		IF	axis_is_standstill(axis)
			AND digital_actuator_is_inactive(csp_transfer_crosspusher_reject.reject_sact)
			AND (
					ABS(axis_calculated_cam_slave_position_deg - slave_scaling) < 2 (* CHECKS IF THE CALCULATED MOVE IS WITHIN 2 mm's OF THE SLAVE SCALING - MEANING AT LOAD *)
					OR csp_transfer_crosspusher.loader_clear (* VERIFIES THE LOADER IS CLEAR MEANING IN A RETRACTED POSITION *)
				)		
		THEN			
			axis_move_absolute(
				position 		:= axis_calculated_cam_slave_position_deg, 
				velocity 		:= phase_velocity_degps,
				direction		:= AXIS_SHORTEST_WAY,
				acceleration 	:= MOTOR_MAX_ACCELLERATION_DEGPS2/4,
				deceleration 	:= MOTOR_MAX_DECELLERATION_DEGPS2/4, 
				jerk 			:= MOTOR_MAX_JERK_DEGPS3, 
				buffer_mode 	:= AXIS_BUFFER_MODE_BUFFERED,
				CONVERSION_this := axis
				);
		END_IF

		IF axis_is_absolute_moving(axis)
		THEN
			phase_status_next	:=	CSP_TRANSFER_PHASE_STATUS_PHASING;
		END_IF

		
	CSP_TRANSFER_PHASE_STATUS_PHASING:

		IF axis_is_standstill(axis)
		THEN
			phase_status_next	:=	CSP_TRANSFER_CROSSPUSHER_STATUS_PHASED;
		END_IF

		
	CSP_TRANSFER_CROSSPUSHER_STATUS_PHASED:

		IF engage_enable
		THEN
			phase_status_next := CSP_TRANSFER_CROSSPUSHER_PHASE_STATUS_DONE;
		END_IF
		
		
	CSP_TRANSFER_CROSSPUSHER_PHASE_STATUS_DONE:	(* Phase done *)
			
		phase_running := FALSE;
		phase_done := TRUE;				
	
		
	CSP_TRANSFER_CROSSPUSHER_PHASE_STATUS_ERROR:	(* Phase error *)
		IF	phase_running
		THEN
			phase_error := TRUE;
			axis_disable(axis);									
		END_IF
		phase_running := FALSE;
		
		IF	phase_conditions 	
		THEN
			phase_status_next := CSP_TRANSFER_CROSSPUSHER_PHASE_STATUS_START;
		END_IF		
END_CASE


IF 	NOT debug_phase_state_machine
	OR debug_phase_machine_one_step	
THEN
	phase_status := phase_status_next;
END_IF

(* Phasing timeout *)
IF (phase_running
	AND NOT debug_phase_state_machine)
	OR phase_error
THEN
	IF	timer_is_expired(phase_time_out_tmr)
	THEN
		process_message_set(1, phase_status, 0, phase_faulted_aem);
	END_IF
ELSE
	timer_restart(30000, phase_time_out_tmr);
END_IF
END_ACTION

END_PROGRAM

// ---- Application/CSP/Case/Closing/csp_case_closing.TcPOU
(*********************************** G.D S.p.A. - Technical Department ***********************************
============= PROGRAM INFO ============
FOLDER:             TBD
MACHINES INVOLVED:  TBD 

============= DESCRIPTION =============
csp machine declaration

============= REVISIONS ===============
Date		Version	 	Author      	Description             
----------	-------		------------  	--------------------------------------------
2019/04/05 	0000.00	 	M.Grasso		Creation of the PRG

**********************************************************************************************************)
(*$R process_ref := prc; $*)
PROGRAM csp_case_closing
VAR
		
	prc:												process;
	prc_path:											STRING;
	RFID_status:										csp_case_closing_rfid_status_enum;
	RFID_status_next:									csp_case_closing_rfid_status_enum;
	
	Closing_RFID_Check_Complete: 						BOOL := FALSE;
	Closing_Upper_RFID_Check_Req: 						BOOL := FALSE;
	
	(* RFID *)
	check_pos_tolerance:								LREAL := 2;
	rfid_value_to_check: 								BYTE;
	os_rfid_value:										BYTE;
	ls_rfid_value:										BYTE;
	
	
	rfid_value_to_write:								BYTE;
	
	(*OS*)
	os_rfid_input_buffer:								iol_slave_bis00lh_pdo_input;
	os_rfid_input_bitheader_1:							iol_slave_bis00lh_bitheader_input;
	os_rfid_input_bitheader_2:							iol_slave_bis00lh_bitheader_input;
			
	os_rfid_output_buffer:								iol_slave_bis00lh_pdo_output;
	os_rfid_output_bitheader_1:							iol_slave_bis00lh_bitheader_output;
	os_rfid_output_bitheader_2:							iol_slave_bis00lh_bitheader_output;
	os_upper_rfid_read_value: 							BYTE;
	os_lower_rfid_read_value: 							BYTE;
	
	(*LS*)
	ls_rfid_input_buffer:								iol_slave_bis00lh_pdo_input;
	ls_rfid_input_bitheader_1:							iol_slave_bis00lh_bitheader_input;
	ls_rfid_input_bitheader_2:							iol_slave_bis00lh_bitheader_input;
			
	ls_rfid_output_buffer:								iol_slave_bis00lh_pdo_output;
	ls_rfid_output_bitheader_1:							iol_slave_bis00lh_bitheader_output;
	ls_rfid_output_bitheader_2:							iol_slave_bis00lh_bitheader_output;
	ls_upper_rfid_read_value: 							BYTE;
	ls_lower_rfid_read_value: 							BYTE;


	rfid_start_toggle:									BOOL := FALSE;
	rfid_shutdown_toggle:								BOOL := FALSE;
	rfid_write_toggle:									BOOL := FALSE;
	rfid_write_done:									BOOL := FALSE;
	rfid_read_toggle:									BOOL := FALSE;
	rfid_read_done:										BOOL := FALSE;
	rfid_read_success: 									BOOL := FALSE;
	Closing_paddle_rfid_error: 							message;

	RFID_read_write_debug: 								BOOL := FALSE;
	RFID_read_write_one_step: 							BOOL := FALSE;
	
	LS_Lower_RFID_Failed: 								message;
	OS_Lower_RFID_Failed: 								message;
	LS_Upper_RFID_Failed: 								message;
	OS_Upper_RFID_Failed: 								message;
	
	RFID_read_bypass: 									BOOL;	//added 05/17/21 PRS	
	
	OS_Closing_Paddles_cleanout_position:				BOOL := FALSE; (*$P $*)
	ClosingRfidCheckVel:								REAL := 10;
	
END_VAR

VAR CONSTANT
	MOTOR_MAX_VELOCITY_DEGPS:							LREAL := 9600;
	MOTOR_MAX_ACCELLERATION_DEGPS2:						LREAL := 4800;
	MOTOR_MAX_DECELLERATION_DEGPS2:						LREAL := 4800;
	MOTOR_MAX_JERK_DEGPS3:								LREAL := 100000000; 
	MOTOR_MAX_FOLLOWING_ERROR_DEG:						LREAL := 2;
END_VAR

_read_var_input();

_object_manager();

IF NOT objects_running()
THEN
	RETURN;	
END_IF

_read_process_image();

_mode_manager();

_set_runtime_properties();

(********************************* BODY *********************************)
IF csp_main_accuChange.RFID_reader_list_accuchange = CLOSING_PADDLES_READER
THEN
	RFID();
END_IF
IF
	( 
	NOT csp_main_accuChange.RFID_read_write_running
	AND (RFID_status = CSP_CASE_CLOSING_RFID_STATUS_COMPLETE 
	OR RFID_status = CSP_CASE_CLOSING_RFID_STATUS_ERROR) 
	)	
THEN
	RFID_status_next := CSP_CASE_CLOSING_RFID_STATUS_START;
END_IF
IF csp_main_accuChange.RFID_check_request AND Closing_RFID_Check_Complete 
THEN
	Closing_RFID_Check_Complete := FALSE;
END_IF
IF csp_main_accuChange.RFID_writing 
	OR csp_main_accuChange.RFID_reading
THEN
	CASE RFID_status OF
		
		CSP_CASE_CLOSING_RFID_STATUS_START:
		
			rfid_read_done := FALSE;
			rfid_write_done := FALSE;
			
			rfid_value_to_write := csp_main_accuchange.RFID_Setup_write_value;
		
			IF 	machine_is_ready(csp.mch)
			THEN
				axis_enable(csp_case_closing_ls_horizontal.axis);
				axis_enable(csp_case_closing_os_horizontal.axis);
				axis_enable(csp_case_closing_ls_lower.axis);
				axis_enable(csp_case_closing_ls_upper.axis);
				axis_enable(csp_case_closing_os_lower.axis);
				axis_enable(csp_case_closing_os_upper.axis);
				RFID_status_next := CSP_CASE_CLOSING_RFID_STATUS_ENABLED;
			END_IF
			
		CSP_CASE_CLOSING_RFID_STATUS_ENABLED:
			
						
			IF 	axis_is_standstill(csp_case_closing_ls_horizontal.axis)
				AND axis_is_standstill(csp_case_closing_os_horizontal.axis)
				AND axis_is_standstill(csp_case_closing_ls_lower.axis)
				AND axis_is_standstill(csp_case_closing_ls_upper.axis)
				AND axis_is_standstill(csp_case_closing_os_lower.axis)
				AND axis_is_standstill(csp_case_closing_os_upper.axis)
			THEN
				axis_move_absolute(
					position 		:= csp_case_closing_ls_horizontal.accu_safe_pos,
					velocity 		:= ClosingRfidCheckVel,
					direction		:= AXIS_SHORTEST_WAY,
					acceleration 	:= MOTOR_MAX_ACCELLERATION_DEGPS2 / 10,
					deceleration 	:= MOTOR_MAX_DECELLERATION_DEGPS2 / 10,
					jerk 			:= MOTOR_MAX_JERK_DEGPS3, 
					buffer_mode 	:= AXIS_BUFFER_MODE_BUFFERED,
					CONVERSION_this := csp_case_closing_ls_horizontal.axis); 
				axis_move_absolute(
					position 		:= csp_case_closing_os_horizontal.accu_safe_pos,
					velocity 		:= ClosingRfidCheckVel,
					direction		:= AXIS_SHORTEST_WAY,
					acceleration 	:= MOTOR_MAX_ACCELLERATION_DEGPS2 / 10,
					deceleration 	:= MOTOR_MAX_DECELLERATION_DEGPS2 / 10,
					jerk 			:= MOTOR_MAX_JERK_DEGPS3, 
					buffer_mode 	:= AXIS_BUFFER_MODE_BUFFERED,
					CONVERSION_this := csp_case_closing_os_horizontal.axis); 			
			END_IF;				
					
			IF 	axis_is_absolute_moving(csp_case_closing_os_horizontal.axis) 
				AND axis_is_absolute_moving(csp_case_closing_ls_horizontal.axis)
			THEN
				RFID_status_next := CSP_CASE_CLOSING_RFID_STATUS_PADDLES_START;
			END_IF				
		
			
		CSP_CASE_CLOSING_RFID_STATUS_PADDLES_START://requests upper paddle to move to rfid check position
			
			IF 	csp_main_accuChange.closing_horizontal_safe // AND csp_main_accuchange.Case_Motors_Safe_accU
				AND axis_is_standstill(csp_case_closing_ls_horizontal.axis)
				AND axis_is_standstill(csp_case_closing_os_horizontal.axis)
			THEN
				Closing_Upper_RFID_Check_Req := TRUE;
				axis_move_absolute(
					position         := csp_case_closing_os_upper.accu_safe_pos, //highest point of paddle
					velocity         := ClosingRfidCheckVel,
					direction        := AXIS_SHORTEST_WAY,
					acceleration     := MOTOR_MAX_ACCELLERATION_DEGPS2 / 10,
					deceleration     := MOTOR_MAX_DECELLERATION_DEGPS2 / 10,
					jerk             := MOTOR_MAX_JERK_DEGPS3,
					buffer_mode     := AXIS_BUFFER_MODE_BUFFERED,
					CONVERSION_this := csp_case_closing_os_upper.axis);  
					
				axis_move_absolute(
					position         := csp_case_closing_ls_upper.accu_safe_pos, //highest point of paddle
					velocity         := ClosingRfidCheckVel*0.76,
					direction        := AXIS_SHORTEST_WAY,
					acceleration     := MOTOR_MAX_ACCELLERATION_DEGPS2 / 10,
					deceleration     := MOTOR_MAX_DECELLERATION_DEGPS2 / 10,
					jerk             := MOTOR_MAX_JERK_DEGPS3,
					buffer_mode     := AXIS_BUFFER_MODE_BUFFERED,
					CONVERSION_this := csp_case_closing_ls_upper.axis);  
				axis_move_absolute(
					position         := csp_case_closing_os_lower.accu_safe_pos, //lowest point of paddle
					velocity         := ClosingRfidCheckVel,
					direction        := AXIS_SHORTEST_WAY,
					acceleration     := MOTOR_MAX_ACCELLERATION_DEGPS2 / 10,
					deceleration     := MOTOR_MAX_DECELLERATION_DEGPS2 / 10,
					jerk             := MOTOR_MAX_JERK_DEGPS3,
					buffer_mode     := AXIS_BUFFER_MODE_BUFFERED,
					CONVERSION_this := csp_case_closing_os_lower.axis);  
					
				axis_move_absolute(
					position         := csp_case_closing_ls_lower.accu_safe_pos, //lowest point of paddle
					velocity         := ClosingRfidCheckVel,
					direction        := AXIS_SHORTEST_WAY,
					acceleration     := MOTOR_MAX_ACCELLERATION_DEGPS2 / 10,
					deceleration     := MOTOR_MAX_DECELLERATION_DEGPS2 / 10,
					jerk             := MOTOR_MAX_JERK_DEGPS3,
					buffer_mode     := AXIS_BUFFER_MODE_BUFFERED,
					CONVERSION_this := csp_case_closing_ls_lower.axis);
				
				IF 	(axis_is_absolute_moving(csp_case_closing_ls_upper.axis) OR csp_case_closing_ls_upper.in_accu_safe_pos)
					AND (axis_is_absolute_moving(csp_case_closing_os_upper.axis) OR csp_case_closing_os_upper.in_accu_safe_pos)
					AND (axis_is_absolute_moving(csp_case_closing_os_lower.axis) OR csp_case_closing_os_lower.in_accu_safe_pos)
					AND (axis_is_absolute_moving(csp_case_closing_ls_lower.axis) OR csp_case_closing_ls_lower.in_accu_safe_pos)
				THEN
					RFID_status_next := CSP_CASE_CLOSING_RFID_STATUS_VERIFY_AXIS_SAFE_POS;
				END_IF
			END_IF
		
			
		CSP_CASE_CLOSING_RFID_STATUS_VERIFY_AXIS_SAFE_POS:	
		
			IF 	csp_case_closing_ls_upper.in_accu_safe_pos
				AND csp_case_closing_os_upper.in_accu_safe_pos
				AND csp_case_closing_os_lower.in_accu_safe_pos
				AND csp_case_closing_ls_lower.in_accu_safe_pos
				AND axis_is_standstill(csp_case_closing_ls_lower.axis)
				AND axis_is_standstill(csp_case_closing_ls_upper.axis)
				AND axis_is_standstill(csp_case_closing_os_lower.axis)
				AND axis_is_standstill(csp_case_closing_os_upper.axis)
			THEN
				RFID_status_next := CSP_CASE_CLOSING_RFID_STATUS_UPPER_START;
			END_IF
				
		CSP_CASE_CLOSING_RFID_STATUS_UPPER_START:	
					
			axis_move_absolute(
					position         := csp_case_closing_os_upper.RFID_check_pos, 
					velocity         := ClosingRfidCheckVel,
					direction        := AXIS_SHORTEST_WAY,
					acceleration     := MOTOR_MAX_ACCELLERATION_DEGPS2 / 10,
					deceleration     := MOTOR_MAX_DECELLERATION_DEGPS2 / 10,
					jerk             := MOTOR_MAX_JERK_DEGPS3,
					buffer_mode     := AXIS_BUFFER_MODE_BUFFERED,
					CONVERSION_this := csp_case_closing_os_upper.axis);  
					
				axis_move_absolute(
					position         := csp_case_closing_ls_upper.RFID_check_pos,
					velocity         := ClosingRfidCheckVel*0.76,
					direction        := AXIS_SHORTEST_WAY,
					acceleration     := MOTOR_MAX_ACCELLERATION_DEGPS2 / 10,
					deceleration     := MOTOR_MAX_DECELLERATION_DEGPS2 / 10,
					jerk             := MOTOR_MAX_JERK_DEGPS3,
					buffer_mode     := AXIS_BUFFER_MODE_BUFFERED,
					CONVERSION_this := csp_case_closing_ls_upper.axis);  
			IF axis_is_absolute_moving(csp_case_closing_ls_upper.axis) 
				AND axis_is_absolute_moving(csp_case_closing_os_upper.axis) 
			THEN
				RFID_status_next := CSP_CASE_CLOSING_RFID_STATUS_UPPER_VERIFY_AXIS_POS;
			END_IF
			
		CSP_CASE_CLOSING_RFID_STATUS_UPPER_VERIFY_AXIS_POS:
			
			IF 	(ABS(csp_case_closing_ls_upper.axis.actual_modulo_position - csp_case_closing_ls_upper.rfid_check_pos)) < check_pos_tolerance
				AND
				(ABS(csp_case_closing_os_upper.axis.actual_modulo_position - csp_case_closing_os_upper.rfid_check_pos)) < check_pos_tolerance
				THEN
					RFID_status_next := CSP_CASE_CLOSING_RFID_STATUS_UPPER_READ_START;
			END_IF
		
			
		CSP_CASE_CLOSING_RFID_STATUS_UPPER_READ_START: 
		
			IF 	(
					(
						ls_rfid_input_bitheader_1.CP 
						AND ls_rfid_input_bitheader_2.CP
						AND os_rfid_input_bitheader_1.CP 
						AND os_rfid_input_bitheader_2.CP
					)
					OR RFID_read_bypass
				)  //added 05/17/21 PRS
				AND axis_is_standstill(csp_case_closing_ls_upper.axis)
				AND axis_is_standstill(csp_case_closing_os_upper.axis)
			THEN
				rfid_start_toggle := TRUE; 
				rfid_read_toggle := csp_main_accuchange.RFID_reading;
				rfid_write_toggle := csp_main_accuchange.RFID_writing;
				RFID_status_next := SEL(rfid_read_toggle,CSP_CASE_CLOSING_RFID_STATUS_UPPER_RETURN_TO_SAFE_POS,CSP_CASE_CLOSING_RFID_STATUS_UPPER_READ_CHECK_RESULT);
			END_IF
				
					
		CSP_CASE_CLOSING_RFID_STATUS_UPPER_READ_CHECK_RESULT: //wait for successful read and store values
		
			IF 	rfid_read_success
			THEN
				ls_upper_rfid_read_value := ls_rfid_value;
				os_upper_rfid_read_value := os_rfid_value;
				IF 	ls_rfid_value = os_rfid_value
					OR RFID_read_bypass 
				THEN
					rfid_value_to_check := os_rfid_value;
					RFID_status_next := CSP_CASE_CLOSING_RFID_STATUS_UPPER_RETURN_TO_SAFE_POS;					
				END_IF
			END_IF
			
			
		CSP_CASE_CLOSING_RFID_STATUS_UPPER_RETURN_TO_SAFE_POS:
			
				axis_move_absolute(
					position         := csp_case_closing_os_upper.accu_safe_pos, //highest point of paddle
					velocity         := ClosingRfidCheckVel,
					direction        := AXIS_SHORTEST_WAY,
					acceleration     := MOTOR_MAX_ACCELLERATION_DEGPS2 / 10,
					deceleration     := MOTOR_MAX_DECELLERATION_DEGPS2 / 10,
					jerk             := MOTOR_MAX_JERK_DEGPS3,
					buffer_mode     := AXIS_BUFFER_MODE_BUFFERED,
					CONVERSION_this := csp_case_closing_os_upper.axis);  
					
				axis_move_absolute(
					position         := csp_case_closing_ls_upper.accu_safe_pos, //highest point of paddle
					velocity         := ClosingRfidCheckVel*0.76,
					direction        := AXIS_SHORTEST_WAY,
					acceleration     := MOTOR_MAX_ACCELLERATION_DEGPS2 / 10,
					deceleration     := MOTOR_MAX_DECELLERATION_DEGPS2 / 10,
					jerk             := MOTOR_MAX_JERK_DEGPS3,
					buffer_mode     := AXIS_BUFFER_MODE_BUFFERED,
					CONVERSION_this := csp_case_closing_ls_upper.axis); 
					
				IF 	axis_is_absolute_moving(csp_case_closing_ls_upper.axis) 
					AND axis_is_absolute_moving(csp_case_closing_os_upper.axis) 
				THEN
					RFID_status_next := CSP_CASE_CLOSING_RFID_STATUS_UPPER_READ_DONE;
				END_IF						
			
			
		CSP_CASE_CLOSING_RFID_STATUS_UPPER_READ_DONE://upper has been checked, and is clear to return to safe pos. waits until uppers moved back to safe position
		
			IF csp_case_closing_ls_upper.in_accu_safe_pos 
				AND csp_case_closing_os_upper.in_accu_safe_pos
			THEN
				RFID_status_next := CSP_CASE_CLOSING_RFID_STATUS_LOWER_START;
			END_IF
			
		CSP_CASE_CLOSING_RFID_STATUS_LOWER_START:	
					
			axis_move_absolute(
					position         := csp_case_closing_os_LOWER.RFID_check_pos, 
					velocity         := ClosingRfidCheckVel,
					direction        := AXIS_SHORTEST_WAY,
					acceleration     := MOTOR_MAX_ACCELLERATION_DEGPS2 / 10,
					deceleration     := MOTOR_MAX_DECELLERATION_DEGPS2 / 10,
					jerk             := MOTOR_MAX_JERK_DEGPS3,
					buffer_mode     := AXIS_BUFFER_MODE_BUFFERED,
					CONVERSION_this := csp_case_closing_os_lower.axis);  
					
				axis_move_absolute(
					position         := csp_case_closing_ls_lower.RFID_check_pos,
					velocity         := ClosingRfidCheckVel,
					direction        := AXIS_SHORTEST_WAY,
					acceleration     := MOTOR_MAX_ACCELLERATION_DEGPS2 / 10,
					deceleration     := MOTOR_MAX_DECELLERATION_DEGPS2 / 10,
					jerk             := MOTOR_MAX_JERK_DEGPS3,
					buffer_mode      := AXIS_BUFFER_MODE_BUFFERED,
					CONVERSION_this := csp_case_closing_ls_lower.axis);  
				IF axis_is_absolute_moving(csp_case_closing_ls_lower.axis) 
					AND axis_is_absolute_moving(csp_case_closing_os_LOWER.axis) 
				THEN
					RFID_status_next := CSP_CASE_CLOSING_RFID_STATUS_LOWER_VERIFY_AXIS_POS;
				END_IF
				
		CSP_CASE_CLOSING_RFID_STATUS_LOWER_VERIFY_AXIS_POS:
			
			IF 	ABS(csp_case_closing_os_LOWER.axis.actual_modulo_position - csp_case_closing_os_LOWER.rfid_check_pos) < check_pos_tolerance
				AND
				ABS(csp_case_closing_ls_lower.axis.actual_modulo_position - csp_case_closing_ls_lower.rfid_check_pos) < check_pos_tolerance
				
			THEN
				RFID_status_next := CSP_CASE_CLOSING_RFID_STATUS_LOWER_READ_START;
			END_IF
		
			
		CSP_CASE_CLOSING_RFID_STATUS_LOWER_READ_START: 
		
			IF (
					(
						ls_rfid_input_bitheader_1.CP 
						AND ls_rfid_input_bitheader_2.CP
						AND os_rfid_input_bitheader_1.CP 
						AND os_rfid_input_bitheader_2.CP
					)
					OR RFID_read_bypass
				)
				AND axis_is_standstill(csp_case_closing_os_LOWER.axis)
				AND axis_is_standstill(csp_case_closing_ls_LOWER.axis)
			THEN
				rfid_start_toggle := TRUE; 
				rfid_read_toggle := csp_main_accuchange.RFID_reading;
				rfid_write_toggle := csp_main_accuchange.RFID_writing;
				RFID_status_next := SEL(rfid_read_toggle,CSP_CASE_CLOSING_RFID_STATUS_LOWER_RETURN_TO_SAFE_POS,CSP_CASE_CLOSING_RFID_STATUS_LOWER_READ_CHECK_RESULT);
			END_IF
				
					
		CSP_CASE_CLOSING_RFID_STATUS_LOWER_READ_CHECK_RESULT: //wait for successful read and store values
		
			IF rfid_read_success
			THEN
				ls_lower_rfid_read_value := ls_rfid_value;
				os_lower_rfid_read_value := os_rfid_value;
				IF ls_rfid_value = os_rfid_value
				THEN
					rfid_value_to_check := os_rfid_value;
					RFID_status_next := CSP_CASE_CLOSING_RFID_STATUS_LOWER_RETURN_TO_SAFE_POS;
				END_IF
			END_IF
			
		CSP_CASE_CLOSING_RFID_STATUS_LOWER_RETURN_TO_SAFE_POS:
			
				axis_move_absolute(
					position         := csp_case_closing_os_lower.accu_safe_pos, //highest point of paddle
					velocity         := ClosingRfidCheckVel,
					direction        := AXIS_SHORTEST_WAY,
					acceleration     := MOTOR_MAX_ACCELLERATION_DEGPS2 / 10,
					deceleration     := MOTOR_MAX_DECELLERATION_DEGPS2 / 10,
					jerk             := MOTOR_MAX_JERK_DEGPS3,
					buffer_mode     := AXIS_BUFFER_MODE_BUFFERED,
					CONVERSION_this := csp_case_closing_os_lower.axis);  
					
				axis_move_absolute(
					position         := csp_case_closing_ls_lower.accu_safe_pos, //highest point of paddle
					velocity         := ClosingRfidCheckVel,
					direction        := AXIS_SHORTEST_WAY,
					acceleration     := MOTOR_MAX_ACCELLERATION_DEGPS2 / 10,
					deceleration     := MOTOR_MAX_DECELLERATION_DEGPS2 / 10,
					jerk             := MOTOR_MAX_JERK_DEGPS3,
					buffer_mode     := AXIS_BUFFER_MODE_BUFFERED,
					CONVERSION_this := csp_case_closing_ls_lower.axis); 
					
				IF 	axis_is_absolute_moving(csp_case_closing_os_lower.axis) 
					AND axis_is_absolute_moving(csp_case_closing_ls_lower.axis) 
				THEN
					RFID_status_next := CSP_CASE_CLOSING_RFID_STATUS_LOWER_READ_DONE;
				END_IF						
			
			
		CSP_CASE_CLOSING_RFID_STATUS_LOWER_READ_DONE://upper has been checked, and is clear to return to safe pos. waits until uppers moved back to safe position
		
			IF	csp_case_closing_ls_lower.in_accu_safe_pos 
				AND csp_case_closing_os_lower.in_accu_safe_pos
			THEN
				RFID_status_next := SEL(rfid_read_toggle, CSP_CASE_CLOSING_RFID_STATUS_COMPLETE, CSP_CASE_CLOSING_RFID_STATUS_VERIFY_VALUES);
			END_IF
			
		CSP_CASE_CLOSING_RFID_STATUS_VERIFY_VALUES://checks all four paddles rfid value to be equal
		
			IF ls_lower_rfid_read_value = rfid_value_to_check
				AND os_lower_rfid_read_value = rfid_value_to_check
				AND ls_upper_rfid_read_value = rfid_value_to_check
				AND os_upper_rfid_read_value = rfid_value_to_check
			THEN
				RFID_status_next := CSP_CASE_CLOSING_RFID_STATUS_COMPLETE;
			ELSE
				RFID_status_next := CSP_CASE_CLOSING_RFID_STATUS_ERROR;
			END_IF
			
		CSP_CASE_CLOSING_RFID_STATUS_COMPLETE://checks are complete
		
			rfid_write_done := TRUE;
			rfid_read_done := TRUE;			
			Closing_RFID_Check_Complete := TRUE;
			
		
		CSP_CASE_CLOSING_RFID_STATUS_ERROR: //rfid error
		
			rfid_write_done := TRUE;
			rfid_read_done := TRUE;		
			Closing_RFID_Check_Complete :=FALSE;
			//process_message_set(0,0,0,Closing_paddle_rfid_error); (* Moved to csp_main_accuChange *)
			IF ls_lower_rfid_read_value <> rfid_value_to_check
			THEN
				process_message_set(0,0,0,LS_Lower_RFID_Failed);
			ELSIF os_lower_rfid_read_value <> rfid_value_to_check THEN
				process_message_set(0,0,0,OS_Lower_RFID_Failed);
			ELSIF ls_upper_rfid_read_value <> rfid_value_to_check THEN
				process_message_set(0,0,0,LS_Upper_RFID_Failed);
			ELSIF os_upper_rfid_read_value <> rfid_value_to_check THEN
				process_message_set(0,0,0,OS_Upper_RFID_Failed);
			END_IF
			
	END_CASE
END_IF
(* Resets RFID Failed Messages on Reset  *)
IF machine_get_reset_edge(csp.mch)
THEN
	process_message_reset(LS_Lower_RFID_Failed);
	process_message_reset(OS_Lower_RFID_Failed);
	process_message_reset(LS_Upper_RFID_Failed);
	process_message_reset(OS_Upper_RFID_Failed);
END_IF




(* ADVANCES TO NEXT STEP *)
IF 	NOT RFID_read_write_debug
	OR
	RFID_read_write_one_step	
THEN
	RFID_status := RFID_status_next;
	RFID_read_write_one_step := FALSE;
END_IF
(************************************************************************)

_handle_messages();

_write_output();

ACTION _handle_messages:
;
END_ACTION

ACTION _handle_process_test:
;
END_ACTION

ACTION _mode_manager:
IF process_mode_req_is_pending(prc)
THEN
    process_apply_mode_req_first_step(prc);
    CASE process_get_mode(prc) OF
        MODE_TO_ABSENT:
			;
        MODE_TO_INACTIVE:
			;
        MODE_TO_TEST:
			;
        MODE_TO_OPERATIONAL:
			;
    END_CASE
    process_apply_mode_req_second_step(prc);
END_IF
END_ACTION

ACTION _object_manager:
IF objects_initialization()
THEN
	sub_process_init(
		object_name					:= 'csp_case_closing.prc', 
		process						:= csp_case.prc, 
		CONVERSION_this				:= prc);
		
	prc_path 						:= process_get_path(prc);
	
	process_message_init(
        object_name:= CONCAT(prc_path, 'Closing_paddle_rfid_error'),
        behaviour:= MESSAGE_BEHAVIOUR_STATE,
        reset_timeout:= 0,
        disableable:= TRUE,
        individual_reset:= FALSE,
        machine_reaction:= MACHINE_REACTION_NO_STOP, 
        typology:=  MESSAGE_TYPOLOGY_OBLIGATION, 
        process:= prc,
        CONVERSION_this:= Closing_paddle_rfid_error);
		
	process_message_init(
        object_name:= CONCAT(prc_path, 'LS_Lower_RFID_Failed'),
        behaviour:= MESSAGE_BEHAVIOUR_STATE,
        reset_timeout:= 0,
        disableable:= TRUE,
        individual_reset:= FALSE,
        machine_reaction:= MACHINE_REACTION_NORMAL_STOP, 
        typology:=  MESSAGE_TYPOLOGY_ABNORMAL, 
        process:= prc,
        CONVERSION_this:= LS_Lower_RFID_Failed);

	process_message_init(
        object_name:= CONCAT(prc_path, 'OS_Lower_RFID_Failed'),
        behaviour:= MESSAGE_BEHAVIOUR_STATE,
        reset_timeout:= 0,
        disableable:= TRUE,
        individual_reset:= FALSE,
        machine_reaction:= MACHINE_REACTION_NORMAL_STOP, 
        typology:=  MESSAGE_TYPOLOGY_ABNORMAL, 
        process:= prc,
        CONVERSION_this:= OS_Lower_RFID_Failed);
		
	process_message_init(
        object_name:= CONCAT(prc_path, 'LS_Upper_RFID_Failed'),
        behaviour:= MESSAGE_BEHAVIOUR_STATE,
        reset_timeout:= 0,
        disableable:= TRUE,
        individual_reset:= FALSE,
        machine_reaction:= MACHINE_REACTION_NORMAL_STOP, 
        typology:=  MESSAGE_TYPOLOGY_ABNORMAL, 
        process:= prc,
        CONVERSION_this:= LS_Upper_RFID_Failed);

	process_message_init(
        object_name:= CONCAT(prc_path, 'OS_Upper_RFID_Failed'),
        behaviour:= MESSAGE_BEHAVIOUR_STATE,
        reset_timeout:= 0,
        disableable:= TRUE,
        individual_reset:= FALSE,
        machine_reaction:= MACHINE_REACTION_NORMAL_STOP, 
        typology:=  MESSAGE_TYPOLOGY_ABNORMAL,
        process:= prc,
        CONVERSION_this:= OS_Upper_RFID_Failed);
	
END_IF

IF objects_running()
THEN
	process_cycle(prc);
END_IF
END_ACTION

ACTION _read_process_image:
;
END_ACTION

ACTION _read_var_input:
;
END_ACTION

ACTION _set_runtime_properties:
;
END_ACTION

ACTION _write_output:
;
END_ACTION

ACTION RFID:
(* LS *)
ls_rfid_input_bitheader_1.CP := ls_rfid_input_buffer.ByteArr[0].0;
ls_rfid_input_bitheader_1.AA := ls_rfid_input_buffer.ByteArr[0].1;
ls_rfid_input_bitheader_1.AE := ls_rfid_input_buffer.ByteArr[0].2;
ls_rfid_input_bitheader_1.AF := ls_rfid_input_buffer.ByteArr[0].3;
ls_rfid_input_bitheader_1.Bit4 := ls_rfid_input_buffer.ByteArr[0].4;
ls_rfid_input_bitheader_1._TO := ls_rfid_input_buffer.ByteArr[0].5;
ls_rfid_input_bitheader_1.HF := ls_rfid_input_buffer.ByteArr[0].6;
ls_rfid_input_bitheader_1.BB := ls_rfid_input_buffer.ByteArr[0].7;

ls_rfid_input_bitheader_2.CP := ls_rfid_input_buffer.ByteArr[0].0;
ls_rfid_input_bitheader_2.AA := ls_rfid_input_buffer.ByteArr[0].1;
ls_rfid_input_bitheader_2.AE := ls_rfid_input_buffer.ByteArr[0].2;
ls_rfid_input_bitheader_2.AF := ls_rfid_input_buffer.ByteArr[0].3;
ls_rfid_input_bitheader_2.Bit4 := ls_rfid_input_buffer.ByteArr[0].4;
ls_rfid_input_bitheader_2._TO := ls_rfid_input_buffer.ByteArr[0].5;
ls_rfid_input_bitheader_2.HF := ls_rfid_input_buffer.ByteArr[0].6;
ls_rfid_input_bitheader_2.BB := ls_rfid_input_buffer.ByteArr[0].7;

ls_rfid_output_buffer.ByteArr[0].0 := ls_rfid_output_bitheader_1.AV ;
ls_rfid_output_buffer.ByteArr[0].1 := ls_rfid_output_bitheader_1.Bit1;
ls_rfid_output_buffer.ByteArr[0].2 := ls_rfid_output_bitheader_1.GR;
ls_rfid_output_buffer.ByteArr[0].3 := ls_rfid_output_bitheader_1.Bit3;
ls_rfid_output_buffer.ByteArr[0].4 := ls_rfid_output_bitheader_1.Bit4;
ls_rfid_output_buffer.ByteArr[0].5 := ls_rfid_output_bitheader_1.KA;
ls_rfid_output_buffer.ByteArr[0].6 := ls_rfid_output_bitheader_1.TI;
ls_rfid_output_buffer.ByteArr[0].7 := ls_rfid_output_bitheader_1.Bit7;

ls_rfid_output_buffer.ByteArr[9].0 := ls_rfid_output_bitheader_2.AV ;
ls_rfid_output_buffer.ByteArr[9].1 := ls_rfid_output_bitheader_2.Bit1;
ls_rfid_output_buffer.ByteArr[9].2 := ls_rfid_output_bitheader_2.GR;
ls_rfid_output_buffer.ByteArr[9].3 := ls_rfid_output_bitheader_2.Bit3;
ls_rfid_output_buffer.ByteArr[9].4 := ls_rfid_output_bitheader_2.Bit4;
ls_rfid_output_buffer.ByteArr[9].5 := ls_rfid_output_bitheader_2.KA;
ls_rfid_output_buffer.ByteArr[9].6 := ls_rfid_output_bitheader_2.TI;
ls_rfid_output_buffer.ByteArr[9].7 := ls_rfid_output_bitheader_2.Bit7;


(* OS *)
os_rfid_input_bitheader_1.CP := os_rfid_input_buffer.ByteArr[0].0;
os_rfid_input_bitheader_1.AA := os_rfid_input_buffer.ByteArr[0].1;
os_rfid_input_bitheader_1.AE := os_rfid_input_buffer.ByteArr[0].2;
os_rfid_input_bitheader_1.AF := os_rfid_input_buffer.ByteArr[0].3;
os_rfid_input_bitheader_1.Bit4 := os_rfid_input_buffer.ByteArr[0].4;
os_rfid_input_bitheader_1._TO := os_rfid_input_buffer.ByteArr[0].5;
os_rfid_input_bitheader_1.HF := os_rfid_input_buffer.ByteArr[0].6;
os_rfid_input_bitheader_1.BB := os_rfid_input_buffer.ByteArr[0].7;

os_rfid_input_bitheader_2.CP := os_rfid_input_buffer.ByteArr[0].0;
os_rfid_input_bitheader_2.AA := os_rfid_input_buffer.ByteArr[0].1;
os_rfid_input_bitheader_2.AE := os_rfid_input_buffer.ByteArr[0].2;
os_rfid_input_bitheader_2.AF := os_rfid_input_buffer.ByteArr[0].3;
os_rfid_input_bitheader_2.Bit4 := os_rfid_input_buffer.ByteArr[0].4;
os_rfid_input_bitheader_2._TO := os_rfid_input_buffer.ByteArr[0].5;
os_rfid_input_bitheader_2.HF := os_rfid_input_buffer.ByteArr[0].6;
os_rfid_input_bitheader_2.BB := os_rfid_input_buffer.ByteArr[0].7;

os_rfid_output_buffer.ByteArr[0].0 := os_rfid_output_bitheader_1.AV ;
os_rfid_output_buffer.ByteArr[0].1 := os_rfid_output_bitheader_1.Bit1;
os_rfid_output_buffer.ByteArr[0].2 := os_rfid_output_bitheader_1.GR;
os_rfid_output_buffer.ByteArr[0].3 := os_rfid_output_bitheader_1.Bit3;
os_rfid_output_buffer.ByteArr[0].4 := os_rfid_output_bitheader_1.Bit4;
os_rfid_output_buffer.ByteArr[0].5 := os_rfid_output_bitheader_1.KA;
os_rfid_output_buffer.ByteArr[0].6 := os_rfid_output_bitheader_1.TI;
os_rfid_output_buffer.ByteArr[0].7 := os_rfid_output_bitheader_1.Bit7;

os_rfid_output_buffer.ByteArr[9].0 := os_rfid_output_bitheader_2.AV ;
os_rfid_output_buffer.ByteArr[9].1 := os_rfid_output_bitheader_2.Bit1;
os_rfid_output_buffer.ByteArr[9].2 := os_rfid_output_bitheader_2.GR;
os_rfid_output_buffer.ByteArr[9].3 := os_rfid_output_bitheader_2.Bit3;
os_rfid_output_buffer.ByteArr[9].4 := os_rfid_output_bitheader_2.Bit4;
os_rfid_output_buffer.ByteArr[9].5 := os_rfid_output_bitheader_2.KA;
os_rfid_output_buffer.ByteArr[9].6 := os_rfid_output_bitheader_2.TI;
os_rfid_output_buffer.ByteArr[9].7 := os_rfid_output_bitheader_2.Bit7;


IF rfid_start_toggle
THEN
	ls_rfid_output_bitheader_1.GR := FALSE;
	ls_rfid_output_bitheader_1.KA := FALSE;
	ls_rfid_output_bitheader_1.AV := FALSE;
	ls_rfid_output_bitheader_2.GR := FALSE;
	ls_rfid_output_bitheader_2.KA := FALSE;
	ls_rfid_output_bitheader_2.AV := FALSE;
	
	os_rfid_output_bitheader_1.GR := FALSE;
	os_rfid_output_bitheader_1.KA := FALSE;
	os_rfid_output_bitheader_1.AV := FALSE;
	os_rfid_output_bitheader_2.GR := FALSE;
	os_rfid_output_bitheader_2.KA := FALSE;
	os_rfid_output_bitheader_2.AV := FALSE;
	
	rfid_start_toggle := FALSE;
END_IF

IF rfid_shutdown_toggle
THEN
	ls_rfid_output_bitheader_1.KA := TRUE;
	ls_rfid_output_bitheader_2.KA := TRUE;
	
	os_rfid_output_bitheader_1.KA := TRUE;
	os_rfid_output_bitheader_2.KA := TRUE;
		
	IF 	ls_rfid_input_bitheader_1.HF
		AND ls_rfid_input_bitheader_2.HF
	
		AND os_rfid_input_bitheader_1.HF
		AND os_rfid_input_bitheader_2.HF
	
		AND NOT ls_rfid_input_bitheader_1.CP
		AND NOT ls_rfid_input_bitheader_2.CP
	
		AND NOT os_rfid_input_bitheader_1.CP
		AND NOT os_rfid_input_bitheader_2.CP
	THEN
		ls_rfid_output_bitheader_1.KA := FALSE;
		ls_rfid_output_bitheader_2.KA := FALSE;
		
		os_rfid_output_bitheader_1.KA := FALSE;
		os_rfid_output_bitheader_2.KA := FALSE;
		
		rfid_shutdown_toggle := FALSE;
	END_IF	
END_IF

IF rfid_write_toggle //OR i_rfid_write_from_hmi
THEN	
	ls_rfid_output_buffer.ByteArr[1] := 16#0032;
	ls_rfid_output_buffer.ByteArr[2] := 16#00;
	ls_rfid_output_buffer.ByteArr[3] := 16#00;
	ls_rfid_output_buffer.ByteArr[4] := 16#0001;
	ls_rfid_output_buffer.ByteArr[5] := 16#00;
	ls_rfid_output_buffer.ByteArr[6] := rfid_value_to_write;
	
	os_rfid_output_buffer.ByteArr[1] := 16#0032;
	os_rfid_output_buffer.ByteArr[2] := 16#00;
	os_rfid_output_buffer.ByteArr[3] := 16#00;
	os_rfid_output_buffer.ByteArr[4] := 16#0001;
	os_rfid_output_buffer.ByteArr[5] := 16#00;
	os_rfid_output_buffer.ByteArr[6] := rfid_value_to_write;
	
	ls_rfid_output_bitheader_1.AV := TRUE;
	ls_rfid_output_bitheader_2.AV := TRUE;
	
	os_rfid_output_bitheader_1.AV := TRUE;
	os_rfid_output_bitheader_2.AV := TRUE;
	
	IF ls_rfid_input_bitheader_1.AA 
		AND ls_rfid_input_bitheader_2.AA 
		AND ls_rfid_input_bitheader_1.AE
		AND ls_rfid_input_bitheader_2.AE
		
		AND os_rfid_input_bitheader_1.AA 
		AND os_rfid_input_bitheader_2.AA 
		AND os_rfid_input_bitheader_1.AE
		AND os_rfid_input_bitheader_2.AE
	THEN
		ls_rfid_output_bitheader_1.AV := FALSE;
		ls_rfid_output_bitheader_2.AV := FALSE;
		
		os_rfid_output_bitheader_1.AV := FALSE;
		os_rfid_output_bitheader_2.AV := FALSE;
		
		rfid_write_toggle := FALSE;
	END_IF		
END_IF

IF rfid_read_toggle 
THEN
	rfid_read_success := FALSE;	
	ls_rfid_output_buffer.ByteArr[1] := 16#0001;
	ls_rfid_output_buffer.ByteArr[2] := 16#00;
	ls_rfid_output_buffer.ByteArr[3] := 16#00;
	ls_rfid_output_buffer.ByteArr[4] := 16#0001;
	ls_rfid_output_buffer.ByteArr[5] := 16#00;
	
	os_rfid_output_buffer.ByteArr[1] := 16#0001;
	os_rfid_output_buffer.ByteArr[2] := 16#00;
	os_rfid_output_buffer.ByteArr[3] := 16#00;
	os_rfid_output_buffer.ByteArr[4] := 16#0001;
	os_rfid_output_buffer.ByteArr[5] := 16#00;
	
	ls_rfid_output_bitheader_1.AV := TRUE;
	ls_rfid_output_bitheader_2.AV := TRUE;
	ls_rfid_value := 0;
	
	os_rfid_output_bitheader_1.AV := TRUE;
	os_rfid_output_bitheader_2.AV := TRUE;
	os_rfid_value := 0;
	
	IF ls_rfid_input_bitheader_1.AA 
		AND ls_rfid_input_bitheader_2.AA 
		AND ls_rfid_input_bitheader_1.AE
		AND ls_rfid_input_bitheader_2.AE
		
		AND os_rfid_input_bitheader_1.AA 
		AND os_rfid_input_bitheader_2.AA 
		AND os_rfid_input_bitheader_1.AE
		AND os_rfid_input_bitheader_2.AE
	THEN
		// SAVE VALUES IN INPUT BUFFER [1...8] - CHECK WITH BRAND FOR WHAT VALUE SHOULD BE PRESENT
		ls_rfid_value := ls_rfid_input_buffer.ByteArr[1];
		ls_rfid_output_bitheader_1.AV := FALSE;
		ls_rfid_output_bitheader_2.AV := FALSE;
		
		os_rfid_value := os_rfid_input_buffer.ByteArr[1];
		os_rfid_output_bitheader_1.AV := FALSE;
		os_rfid_output_bitheader_2.AV := FALSE;
		
		IF ls_rfid_value <> 0 AND os_rfid_value <> 0
		THEN
			rfid_read_success := TRUE;
		END_IF
		rfid_read_toggle := FALSE;
	END_IF		
END_IF
END_ACTION

END_PROGRAM

// ---- Application/CSP/Case/Main/Drives/csp_case_main_drives.TcPOU

(*********************************** G.D S.p.A. - Technical Department ***********************************
============= PROGRAM INFO ============
FOLDER:             TBD
MACHINES INVOLVED:  TBD 

============= DESCRIPTION =============

============= REVISIONS ===============
Date		Version	 	Author      	Description             
----------	-------		------------  	--------------------------------------------
2019/04/24 	0000.00	 	M.Grasso		Creation of the PRG

**********************************************************************************************************)
(*$R 
	process_ref:= prc; 
$*)
PROGRAM csp_case_main_drives
VAR
	prc:						process;
	prc_path:					STRING;	
	
	PS2000_ps:					power_supply;
	
	SD2100_drv:					soe_drive;
	SD2200_drv:					soe_drive;
	SD2300_drv:					soe_drive;
	SD2400_drv:					soe_drive;
	SD2500_drv:					soe_drive;
	
	SD12000_drv:				soe_drive;
	SD8000_drv:					soe_drive;
	SD8100_drv:					soe_drive;
	SD8200_drv:					soe_drive;
	SD8300_drv:					soe_drive;
	SD8400_drv:					soe_drive;
	SD8500_drv:					soe_drive;
	SD8600_drv:					soe_drive;
	
	SD10000_drv:				soe_drive;
	SD10100_drv:				soe_drive;
	SD10200_drv:				soe_drive;
	SD10300_drv:				soe_drive;
	SD10400_drv:				soe_drive;
	SD11000_drv:				soe_drive;
	
	SD15000_drv:				soe_drive;
	
	SD26000_drv:				soe_drive;
	SD26100_drv:				soe_drive;
	
END_VAR

VAR CONSTANT
	INCOHERENCE_TIMEOUT_MS:		DINT := 2000;
END_VAR

_read_var_input();

_objects_manager();

IF NOT objects_running()
THEN
	RETURN;	
END_IF

_read_process_image();

_mode_manager();

CASE process_get_mode(prc) OF
	MODE_ABSENT,
	MODE_INACTIVE:
		RETURN;
	MODE_TEST:
		;
END_CASE

_set_runtime_properties();

(********************************* BODY *********************************)

(************************************************************************)

_handle_messages();

_write_output();

ACTION _handle_messages:
;
END_ACTION

ACTION _handle_process_test:
;
END_ACTION

ACTION _mode_manager:
IF process_mode_req_is_pending(prc)
THEN
    process_apply_mode_req_first_step(prc);
    CASE process_get_mode(prc) OF
        MODE_TO_ABSENT:
			;
        MODE_TO_INACTIVE:
			;
        MODE_TO_TEST:
			;
        MODE_TO_OPERATIONAL:
			;
    END_CASE
    process_apply_mode_req_second_step(prc);
END_IF
END_ACTION

ACTION _objects_manager:
IF objects_initialization()
THEN
	sub_process_init(
		object_name					:= 'csp_case_main_drives.prc', 
		process						:= csp_case_main.prc, 
		CONVERSION_this				:= prc);
		
	prc_path 						:= process_get_path(prc);

	(* PS2000 POWER SUPPLY *)
	power_supply_init(
		object_name					:= CONCAT(prc_path, '_PS2000_ps'), 
		vendor						:= DRIVE_BOSCH_REXROTH, 
		process						:= prc, 
		CONVERSION_this				:= PS2000_ps);
		
	power_supply_add_safety_integrated_series(
		safety_integrated_series	:= csp_case_main_safety_drives_PS2000.sis, 
		CONVERSION_this				:= PS2000_ps);		

		(* SD2100 *)
	soe_drive_double_channel_init(
		object_name					:= CONCAT(prc_path, '_SD2100_drv'), 
		device_name					:= 'SD2100', 
		vendor						:= DRIVE_BOSCH_REXROTH, 
		standalone					:= FALSE, 
		channel_a_name				:= 'csp_case_transport_os_leading_axis', 
		channel_b_name				:= 'csp_case_transport_os_trailing_axis', 
		ethercat_master				:= csp_main.cabinet_ethercat_master, 
		process						:= prc, 
		CONVERSION_this				:= SD2100_drv);	
		
	soe_drive_add_power_supply(
		power_supply				:= PS2000_ps, 
		CONVERSION_this				:= SD2100_drv);
		
	IF 	SD2100_drv.channel_a.has_channel
	THEN	
		soe_drive_enable_fsoe(
			handler						:= BOSCH_DRIVE_CHANNEL_A, 
			incoherence_timeout			:= INCOHERENCE_TIMEOUT_MS, 
			connection_interface		:= csp_case_main_safety_interface._SD2100_drv_ChA, 
			group						:= csp_case_main_safety_drives_SD2100.sig, 
			CONVERSION_this				:= SD2100_drv);
	END_IF
		
	IF 	SD2100_drv.channel_B.has_channel
	THEN	
		soe_drive_enable_fsoe(
			handler						:= BOSCH_DRIVE_CHANNEL_B, 
			incoherence_timeout			:= INCOHERENCE_TIMEOUT_MS, 
			connection_interface		:= csp_case_main_safety_interface._SD2100_drv_ChB, 
			group						:= csp_case_main_safety_drives_SD2100.sig, 
			CONVERSION_this				:= SD2100_drv);
	END_IF
	
	(* SD2200 *)
	soe_drive_double_channel_init(
		object_name					:= CONCAT(prc_path, '_SD2200_drv'), 
		device_name					:= 'SD2200', 
		vendor						:= DRIVE_BOSCH_REXROTH, 
		standalone					:= FALSE, 
		channel_a_name				:= 'csp_case_transport_ls_leading_axis', 
		channel_b_name				:= 'csp_case_transport_ls_trailing_axis', 
		ethercat_master				:= csp_main.cabinet_ethercat_master, 
		process						:= prc, 
		CONVERSION_this				:= SD2200_drv);	
		
	soe_drive_add_power_supply(
		power_supply				:= PS2000_ps, 
		CONVERSION_this				:= SD2200_drv);
		
	IF 	SD2200_drv.channel_a.has_channel
	THEN	
		soe_drive_enable_fsoe(
			handler						:= BOSCH_DRIVE_CHANNEL_A, 
			incoherence_timeout			:= INCOHERENCE_TIMEOUT_MS, 
			connection_interface		:= csp_case_main_safety_interface._SD2200_drv_ChA, 
			group						:= csp_case_main_safety_drives_SD2200.sig, 
			CONVERSION_this				:= SD2200_drv);
	END_IF
		
	IF 	SD2200_drv.channel_B.has_channel
	THEN	
		soe_drive_enable_fsoe(
			handler						:= BOSCH_DRIVE_CHANNEL_B, 
			incoherence_timeout			:= INCOHERENCE_TIMEOUT_MS, 
			connection_interface		:= csp_case_main_safety_interface._SD2200_drv_ChB, 
			group						:= csp_case_main_safety_drives_SD2200.sig, 
			CONVERSION_this				:= SD2200_drv);
	END_IF
	
	(* SD2300 *)
	soe_drive_double_channel_init(
		object_name					:= CONCAT(prc_path, '_SD2300_drv'), 
		device_name					:= 'SD2300', 
		vendor						:= DRIVE_BOSCH_REXROTH, 
		standalone					:= FALSE, 
		channel_a_name				:= 'csp_case_closing_os_upper_axis', 
		channel_b_name				:= 'csp_case_closing_os_lower_axis', 
		ethercat_master				:= csp_main.cabinet_ethercat_master, 
		process						:= prc, 
		CONVERSION_this				:= SD2300_drv);	
		
	soe_drive_add_power_supply(
		power_supply				:= PS2000_ps, 
		CONVERSION_this				:= SD2300_drv);
		
	IF 	SD2300_drv.channel_a.has_channel
	THEN	
		soe_drive_enable_fsoe(
			handler						:= BOSCH_DRIVE_CHANNEL_A, 
			incoherence_timeout			:= INCOHERENCE_TIMEOUT_MS, 
			connection_interface		:= csp_case_main_safety_interface._SD2300_drv_ChA, 
			group						:= csp_case_main_safety_drives_SD2300.sig, 
			CONVERSION_this				:= SD2300_drv);
	END_IF
		
	IF 	SD2300_drv.channel_B.has_channel
	THEN	
		soe_drive_enable_fsoe(
			handler						:= BOSCH_DRIVE_CHANNEL_B, 
			incoherence_timeout			:= INCOHERENCE_TIMEOUT_MS, 
			connection_interface		:= csp_case_main_safety_interface._SD2300_drv_ChB, 
			group						:= csp_case_main_safety_drives_SD2300.sig, 
			CONVERSION_this				:= SD2300_drv);
	END_IF
	
	(* SD2400 *)
	soe_drive_double_channel_init(
		object_name					:= CONCAT(prc_path, '_SD2400_drv'), 
		device_name					:= 'SD2400', 
		vendor						:= DRIVE_BOSCH_REXROTH, 
		standalone					:= FALSE, 
		channel_a_name				:= 'csp_case_closing_os_horizontal_axis', 
		channel_b_name				:= 'csp_case_closing_ls_upper_axis', 
		ethercat_master				:= csp_main.cabinet_ethercat_master, 
		process						:= prc, 
		CONVERSION_this				:= SD2400_drv);	
		
	soe_drive_add_power_supply(
		power_supply				:= PS2000_ps, 
		CONVERSION_this				:= SD2400_drv);
		
	IF 	SD2400_drv.channel_a.has_channel
	THEN	
		soe_drive_enable_fsoe(
			handler						:= BOSCH_DRIVE_CHANNEL_A, 
			incoherence_timeout			:= INCOHERENCE_TIMEOUT_MS, 
			connection_interface		:= csp_case_main_safety_interface._SD2400_drv_ChA, 
			group						:= csp_case_main_safety_drives_SD2400.sig, 
			CONVERSION_this				:= SD2400_drv);
	END_IF
		
	IF 	SD2400_drv.channel_B.has_channel
	THEN	
		soe_drive_enable_fsoe(
			handler						:= BOSCH_DRIVE_CHANNEL_B, 
			incoherence_timeout			:= INCOHERENCE_TIMEOUT_MS, 
			connection_interface		:= csp_case_main_safety_interface._SD2400_drv_ChB, 
			group						:= csp_case_main_safety_drives_SD2400.sig, 
			CONVERSION_this				:= SD2400_drv);
	END_IF
	
	(* SD2500 *)
	soe_drive_double_channel_init(
		object_name					:= CONCAT(prc_path, '_SD2500_drv'), 
		device_name					:= 'SD2500', 
		vendor						:= DRIVE_BOSCH_REXROTH, 
		standalone					:= FALSE, 
		channel_a_name				:= 'csp_case_closing_ls_lower_axis', 
		channel_b_name				:= 'csp_case_closing_ls_horizontal_axis', 
		ethercat_master				:= csp_main.cabinet_ethercat_master, 
		process						:= prc, 
		CONVERSION_this				:= SD2500_drv);	
		
	soe_drive_add_power_supply(
		power_supply				:= PS2000_ps, 
		CONVERSION_this				:= SD2500_drv);
		
	IF 	SD2500_drv.channel_a.has_channel
	THEN	
		soe_drive_enable_fsoe(
			handler						:= BOSCH_DRIVE_CHANNEL_A, 
			incoherence_timeout			:= INCOHERENCE_TIMEOUT_MS, 
			connection_interface		:= csp_case_main_safety_interface._SD2500_drv_ChA, 
			group						:= csp_case_main_safety_drives_SD2500.sig, 
			CONVERSION_this				:= SD2500_drv);
	END_IF
		
	IF 	SD2500_drv.channel_B.has_channel
	THEN	
		soe_drive_enable_fsoe(
			handler						:= BOSCH_DRIVE_CHANNEL_B, 
			incoherence_timeout			:= INCOHERENCE_TIMEOUT_MS, 
			connection_interface		:= csp_case_main_safety_interface._SD2500_drv_ChB, 
			group						:= csp_case_main_safety_drives_SD2500.sig, 
			CONVERSION_this				:= SD2500_drv);
	END_IF
	
		
		(* SD12000 *)
	soe_drive_double_channel_init(
		object_name					:= CONCAT(prc_path, '_SD12000_drv'), 
		device_name					:= 'SD12000', 
		vendor						:= DRIVE_BOSCH_REXROTH, 
		standalone					:= FALSE, 
		channel_a_name				:= 'csp_case_discharge_speedBelt_os_axis', 
		channel_b_name				:= 'csp_case_discharge_speedBelt_ls_axis', 
		ethercat_master				:= csp_main.cabinet_ethercat_master, 
		process						:= prc, 
		CONVERSION_this				:= SD12000_drv);	
		
	soe_drive_add_power_supply(
		power_supply				:= PS2000_ps, 
		CONVERSION_this				:= SD12000_drv);
		
	IF 	SD12000_drv.channel_a.has_channel
	THEN	
		soe_drive_enable_fsoe(
			handler						:= BOSCH_DRIVE_CHANNEL_A, 
			incoherence_timeout			:= INCOHERENCE_TIMEOUT_MS, 
			connection_interface		:= csp_case_main_safety_interface._SD12000_drv_ChA, 
			group						:= csp_case_main_safety_drives_SD12000.sig, 
			CONVERSION_this				:= SD12000_drv);
	END_IF
		
	IF 	SD12000_drv.channel_B.has_channel
	THEN	
		soe_drive_enable_fsoe(
			handler						:= BOSCH_DRIVE_CHANNEL_B, 
			incoherence_timeout			:= INCOHERENCE_TIMEOUT_MS, 
			connection_interface		:= csp_case_main_safety_interface._SD12000_drv_ChB, 
			group						:= csp_case_main_safety_drives_SD12000.sig, 
			CONVERSION_this				:= SD12000_drv);
	END_IF
	
	(* SD8000 *)
	soe_drive_double_channel_init(
		object_name					:= CONCAT(prc_path, '_SD8000_drv'), 
		device_name					:= 'SD8000', 
		vendor						:= DRIVE_BOSCH_REXROTH, 
		standalone					:= FALSE, 
		channel_a_name				:= 'csp_case_feed_shuttle_horizontal_axis', 
		channel_b_name				:= 'csp_case_feed_shuttle_vertical_axis', 
		ethercat_master				:= csp_main.cabinet_ethercat_master, 
		process						:= prc, 
		CONVERSION_this				:= SD8000_drv);	
		
	soe_drive_add_power_supply(
		power_supply				:= PS2000_ps, 
		CONVERSION_this				:= SD8000_drv);
		
	IF 	SD8000_drv.channel_a.has_channel
	THEN	
		soe_drive_enable_fsoe(
			handler						:= BOSCH_DRIVE_CHANNEL_A, 
			incoherence_timeout			:= INCOHERENCE_TIMEOUT_MS, 
			connection_interface		:= csp_case_main_safety_interface._SD8000_drv_ChA, 
			group						:= csp_case_main_safety_drives_SD8000.sig, 
			CONVERSION_this				:= SD8000_drv);
	END_IF
		
	IF 	SD8000_drv.channel_B.has_channel
	THEN	
		soe_drive_enable_fsoe(
			handler						:= BOSCH_DRIVE_CHANNEL_B, 
			incoherence_timeout			:= INCOHERENCE_TIMEOUT_MS, 
			connection_interface		:= csp_case_main_safety_interface._SD8000_drv_ChB, 
			group						:= csp_case_main_safety_drives_SD8000.sig, 
			CONVERSION_this				:= SD8000_drv);
	END_IF
	
	(* SD8100 *)
	soe_drive_double_channel_init(
		object_name					:= CONCAT(prc_path, '_SD8100_drv'), 
		device_name					:= 'SD8100', 
		vendor						:= DRIVE_BOSCH_REXROTH, 
		standalone					:= FALSE, 
		channel_a_name				:= 'csp_case_feed_arm_shoulder_axis', 
		channel_b_name				:= 'csp_case_fc_ls_lower_trailingCloser_axis', 
		ethercat_master				:= csp_main.cabinet_ethercat_master, 
		process						:= prc, 
		CONVERSION_this				:= SD8100_drv);	
		
	soe_drive_add_power_supply(
		power_supply				:= PS2000_ps, 
		CONVERSION_this				:= SD8100_drv);
		
	IF 	SD8100_drv.channel_a.has_channel
	THEN	
		soe_drive_enable_fsoe(
			handler						:= BOSCH_DRIVE_CHANNEL_A, 
			incoherence_timeout			:= INCOHERENCE_TIMEOUT_MS, 
			connection_interface		:= csp_case_main_safety_interface._SD8100_drv_ChA, 
			group						:= csp_case_main_safety_drives_SD8100.sig, 
			CONVERSION_this				:= SD8100_drv);
	END_IF
		
	IF 	SD8100_drv.channel_B.has_channel
	THEN	
		soe_drive_enable_fsoe(
			handler						:= BOSCH_DRIVE_CHANNEL_B, 
			incoherence_timeout			:= INCOHERENCE_TIMEOUT_MS, 
			connection_interface		:= csp_case_main_safety_interface._SD8100_drv_ChB, 
			group						:= csp_case_main_safety_drives_SD8100.sig, 
			CONVERSION_this				:= SD8100_drv);
	END_IF	
	
	(* SD8200 *)
	soe_drive_double_channel_init(
		object_name					:= CONCAT(prc_path, '_SD8200_drv'), 
		device_name					:= 'SD8200', 
		vendor						:= DRIVE_BOSCH_REXROTH, 
		standalone					:= FALSE, 
		channel_a_name				:= 'csp_case_feed_arm_elbow_axis', 
		channel_b_name				:= 'csp_case_loader_guide_upstream_axis', 
		ethercat_master				:= csp_main.cabinet_ethercat_master, 
		process						:= prc, 
		CONVERSION_this				:= SD8200_drv);	
		
	soe_drive_add_power_supply(
		power_supply				:= PS2000_ps, 
		CONVERSION_this				:= SD8200_drv);
		
	IF 	SD8200_drv.channel_a.has_channel
	THEN	
		soe_drive_enable_fsoe(
			handler						:= BOSCH_DRIVE_CHANNEL_A, 
			incoherence_timeout			:= INCOHERENCE_TIMEOUT_MS, 
			connection_interface		:= csp_case_main_safety_interface._SD8200_drv_ChA, 
			group						:= csp_case_main_safety_drives_SD8200.sig, 
			CONVERSION_this				:= SD8200_drv);
	END_IF
		
	IF 	SD8200_drv.channel_B.has_channel
	THEN	
		soe_drive_enable_fsoe(
			handler						:= BOSCH_DRIVE_CHANNEL_B, 
			incoherence_timeout			:= INCOHERENCE_TIMEOUT_MS, 
			connection_interface		:= csp_case_main_safety_interface._SD8200_drv_ChB, 
			group						:= csp_case_main_safety_drives_SD8200.sig, 
			CONVERSION_this				:= SD8200_drv);
	END_IF	
	
	(* SD8300 *)
	soe_drive_double_channel_init(
		object_name					:= CONCAT(prc_path, '_SD8300_drv'), 
		device_name					:= 'SD8300', 
		vendor						:= DRIVE_BOSCH_REXROTH, 
		standalone					:= FALSE, 
		channel_a_name				:= 'csp_case_feed_arm_wrist_axis', 
		channel_b_name				:= 'csp_case_loader_guide_downstream_axis', 
		ethercat_master				:= csp_main.cabinet_ethercat_master, 
		process						:= prc, 
		CONVERSION_this				:= SD8300_drv);	
		
	soe_drive_add_power_supply(
		power_supply				:= PS2000_ps, 
		CONVERSION_this				:= SD8300_drv);
		
	IF 	SD8300_drv.channel_a.has_channel
	THEN	
		soe_drive_enable_fsoe(
			handler						:= BOSCH_DRIVE_CHANNEL_A, 
			incoherence_timeout			:= INCOHERENCE_TIMEOUT_MS, 
			connection_interface		:= csp_case_main_safety_interface._SD8300_drv_ChA, 
			group						:= csp_case_main_safety_drives_SD8300.sig, 
			CONVERSION_this				:= SD8300_drv);
	END_IF
		
	IF 	SD8300_drv.channel_B.has_channel
	THEN	
		soe_drive_enable_fsoe(
			handler						:= BOSCH_DRIVE_CHANNEL_B, 
			incoherence_timeout			:= INCOHERENCE_TIMEOUT_MS, 
			connection_interface		:= csp_case_main_safety_interface._SD8300_drv_ChB, 
			group						:= csp_case_main_safety_drives_SD8300.sig, 
			CONVERSION_this				:= SD8300_drv);
	END_IF	
	
	(* SD8400 *)
	soe_drive_double_channel_init(
		object_name					:= CONCAT(prc_path, '_SD8400_drv'), 
		device_name					:= 'SD8400', 
		vendor						:= DRIVE_BOSCH_REXROTH, 
		standalone					:= FALSE, 
		channel_a_name				:= 'csp_case_feed_magazine_os_belt_axis', 
		channel_b_name				:= 'csp_case_feed_magazine_ls_belt_axis', 
		ethercat_master				:= csp_main.cabinet_ethercat_master, 
		process						:= prc, 
		CONVERSION_this				:= SD8400_drv);	
		
	soe_drive_add_power_supply(
		power_supply				:= PS2000_ps, 
		CONVERSION_this				:= SD8400_drv);
		
	IF 	SD8400_drv.channel_a.has_channel
	THEN	
		soe_drive_enable_fsoe(
			handler						:= BOSCH_DRIVE_CHANNEL_A, 
			incoherence_timeout			:= INCOHERENCE_TIMEOUT_MS, 
			connection_interface		:= csp_case_main_safety_interface._SD8400_drv_ChA, 
			group						:= csp_case_main_safety_drives_SD8400.sig, 
			CONVERSION_this				:= SD8400_drv);
	END_IF
		
	IF 	SD8400_drv.channel_B.has_channel
	THEN	
		soe_drive_enable_fsoe(
			handler						:= BOSCH_DRIVE_CHANNEL_B, 
			incoherence_timeout			:= INCOHERENCE_TIMEOUT_MS, 
			connection_interface		:= csp_case_main_safety_interface._SD8400_drv_ChB, 
			group						:= csp_case_main_safety_drives_SD8400.sig, 
			CONVERSION_this				:= SD8400_drv);
	END_IF	
	
	(* SD8500 *)
	soe_drive_double_channel_init(
		object_name					:= CONCAT(prc_path, '_SD8500_drv'), 
		device_name					:= 'SD8500', 
		vendor						:= DRIVE_BOSCH_REXROTH, 
		standalone					:= FALSE, 
		channel_a_name				:= 'csp_case_loader_pusher_axis', 
		channel_b_name				:= 'csp_case_loader_guide_length_axis', 
		ethercat_master				:= csp_main.cabinet_ethercat_master, 
		process						:= prc, 
		CONVERSION_this				:= SD8500_drv);	
		
	soe_drive_add_power_supply(
		power_supply				:= PS2000_ps, 
		CONVERSION_this				:= SD8500_drv);
		
	IF 	SD8500_drv.channel_a.has_channel
	THEN	
		soe_drive_enable_fsoe(
			handler						:= BOSCH_DRIVE_CHANNEL_A, 
			incoherence_timeout			:= INCOHERENCE_TIMEOUT_MS, 
			connection_interface		:= csp_case_main_safety_interface._SD8500_drv_ChA, 
			group						:= csp_case_main_safety_drives_SD8500.sig, 
			CONVERSION_this				:= SD8500_drv);
	END_IF
		
	IF 	SD8500_drv.channel_B.has_channel
	THEN	
		soe_drive_enable_fsoe(
			handler						:= BOSCH_DRIVE_CHANNEL_B, 
			incoherence_timeout			:= INCOHERENCE_TIMEOUT_MS, 
			connection_interface		:= csp_case_main_safety_interface._SD8500_drv_ChB, 
			group						:= csp_case_main_safety_drives_SD8500.sig, 
			CONVERSION_this				:= SD8500_drv);
	END_IF	
	
	(* SD8600 *)
	soe_drive_double_channel_init(
		object_name					:= CONCAT(prc_path, '_SD8600_drv'), 
		device_name					:= 'SD8600', 
		vendor						:= DRIVE_BOSCH_REXROTH, 
		standalone					:= FALSE, 
		channel_a_name				:= 'csp_case_feed_reject_belt_upper_axis', 
		channel_b_name				:= 'csp_case_feed_reject_belt_lower_axis', 
		ethercat_master				:= csp_main.cabinet_ethercat_master, 
		process						:= prc, 
		CONVERSION_this				:= SD8600_drv);	
		
	soe_drive_add_power_supply(
		power_supply				:= PS2000_ps, 
		CONVERSION_this				:= SD8600_drv);
		
	IF 	SD8600_drv.channel_a.has_channel
	THEN	
		soe_drive_enable_fsoe(
			handler						:= BOSCH_DRIVE_CHANNEL_A, 
			incoherence_timeout			:= INCOHERENCE_TIMEOUT_MS, 
			connection_interface		:= csp_case_main_safety_interface._SD8600_drv_ChA, 
			group						:= csp_case_main_safety_drives_SD8600.sig, 
			CONVERSION_this				:= SD8600_drv);
	END_IF
		
	IF 	SD8600_drv.channel_B.has_channel
	THEN	
		soe_drive_enable_fsoe(
			handler						:= BOSCH_DRIVE_CHANNEL_B, 
			incoherence_timeout			:= INCOHERENCE_TIMEOUT_MS, 
			connection_interface		:= csp_case_main_safety_interface._SD8600_drv_ChB, 
			group						:= csp_case_main_safety_drives_SD8600.sig, 
			CONVERSION_this				:= SD8600_drv);
	END_IF	
	
	(* SD10000 *)
	soe_drive_double_channel_init(
		object_name					:= CONCAT(prc_path, '_SD10000_drv'), 
		device_name					:= 'SD10000', 
		vendor						:= DRIVE_BOSCH_REXROTH, 
		standalone					:= FALSE, 
		channel_a_name				:= 'csp_case_fc_os_upper_spreader_axis', 
		channel_b_name				:= 'csp_case_fc_os_upper_follower_axis', 
		ethercat_master				:= csp_main.cabinet_ethercat_master, 
		process						:= prc, 
		CONVERSION_this				:= SD10000_drv);	
		
	soe_drive_add_power_supply(
		power_supply				:= PS2000_ps, 
		CONVERSION_this				:= SD10000_drv);
		
	IF 	SD10000_drv.channel_a.has_channel
	THEN	
		soe_drive_enable_fsoe(
			handler						:= BOSCH_DRIVE_CHANNEL_A, 
			incoherence_timeout			:= INCOHERENCE_TIMEOUT_MS, 
			connection_interface		:= csp_case_main_safety_interface._SD10000_drv_ChA, 
			group						:= csp_case_main_safety_drives_SD10000.sig, 
			CONVERSION_this				:= SD10000_drv);
	END_IF
		
	IF 	SD10000_drv.channel_B.has_channel
	THEN	
		soe_drive_enable_fsoe(
			handler						:= BOSCH_DRIVE_CHANNEL_B, 
			incoherence_timeout			:= INCOHERENCE_TIMEOUT_MS, 
			connection_interface		:= csp_case_main_safety_interface._SD10000_drv_ChB, 
			group						:= csp_case_main_safety_drives_SD10000.sig, 
			CONVERSION_this				:= SD10000_drv);
	END_IF	
	
	(* SD10100 *)
	soe_drive_double_channel_init(
		object_name					:= CONCAT(prc_path, '_SD10100_drv'), 
		device_name					:= 'SD10100', 
		vendor						:= DRIVE_BOSCH_REXROTH, 
		standalone					:= FALSE, 
		channel_a_name				:= 'csp_case_fc_os_lower_spreader_axis', 
		channel_b_name				:= 'csp_case_fc_os_lower_follower_axis', 
		ethercat_master				:= csp_main.cabinet_ethercat_master, 
		process						:= prc, 
		CONVERSION_this				:= SD10100_drv);	
		
	soe_drive_add_power_supply(
		power_supply				:= PS2000_ps, 
		CONVERSION_this				:= SD10100_drv);
		
	IF 	SD10100_drv.channel_a.has_channel
	THEN	
		soe_drive_enable_fsoe(
			handler						:= BOSCH_DRIVE_CHANNEL_A, 
			incoherence_timeout			:= INCOHERENCE_TIMEOUT_MS, 
			connection_interface		:= csp_case_main_safety_interface._SD10100_drv_ChA, 
			group						:= csp_case_main_safety_drives_SD10100.sig, 
			CONVERSION_this				:= SD10100_drv);
	END_IF
		
	IF 	SD10100_drv.channel_B.has_channel
	THEN	
		soe_drive_enable_fsoe(
			handler						:= BOSCH_DRIVE_CHANNEL_B, 
			incoherence_timeout			:= INCOHERENCE_TIMEOUT_MS, 
			connection_interface		:= csp_case_main_safety_interface._SD10100_drv_ChB, 
			group						:= csp_case_main_safety_drives_SD10100.sig, 
			CONVERSION_this				:= SD10100_drv);
	END_IF	
	
	(* SD10200 *)
	soe_drive_double_channel_init(
		object_name					:= CONCAT(prc_path, '_SD10200_drv'), 
		device_name					:= 'SD10200', 
		vendor						:= DRIVE_BOSCH_REXROTH, 
		standalone					:= FALSE, 
		channel_a_name				:= '',//'csp_case_fc_os_lower_trailingCloser_axis', 
		channel_b_name				:= 'csp_case_fc_ls_upper_spreader_axis', 
		ethercat_master				:= csp_main.cabinet_ethercat_master, 
		process						:= prc, 
		CONVERSION_this				:= SD10200_drv);	
		
	soe_drive_add_power_supply(
		power_supply				:= PS2000_ps, 
		CONVERSION_this				:= SD10200_drv);
		
	IF 	SD10200_drv.channel_a.has_channel
	THEN	
		soe_drive_enable_fsoe(
			handler						:= BOSCH_DRIVE_CHANNEL_A, 
			incoherence_timeout			:= INCOHERENCE_TIMEOUT_MS, 
			connection_interface		:= csp_case_main_safety_interface._SD10200_drv_ChA, 
			group						:= csp_case_main_safety_drives_SD10200.sig, 
			CONVERSION_this				:= SD10200_drv);
	END_IF
		
	IF 	SD10200_drv.channel_B.has_channel
	THEN	
		soe_drive_enable_fsoe(
			handler						:= BOSCH_DRIVE_CHANNEL_B, 
			incoherence_timeout			:= INCOHERENCE_TIMEOUT_MS, 
			connection_interface		:= csp_case_main_safety_interface._SD10200_drv_ChB, 
			group						:= csp_case_main_safety_drives_SD10200.sig, 
			CONVERSION_this				:= SD10200_drv);
	END_IF

	(* SD10300 *)
	soe_drive_double_channel_init(
		object_name					:= CONCAT(prc_path, '_SD10300_drv'), 
		device_name					:= 'SD10300', 
		vendor						:= DRIVE_BOSCH_REXROTH, 
		standalone					:= FALSE, 
		channel_a_name				:= 'csp_case_fc_ls_upper_follower_axis', 
		channel_b_name				:= 'csp_case_fc_ls_upper_leadingMinorCloser_axis', 
		ethercat_master				:= csp_main.cabinet_ethercat_master, 
		process						:= prc, 
		CONVERSION_this				:= SD10300_drv);	
		
	soe_drive_add_power_supply(
		power_supply				:= PS2000_ps, 
		CONVERSION_this				:= SD10300_drv);
		
	IF 	SD10300_drv.channel_a.has_channel
	THEN	
		soe_drive_enable_fsoe(
			handler						:= BOSCH_DRIVE_CHANNEL_A, 
			incoherence_timeout			:= INCOHERENCE_TIMEOUT_MS, 
			connection_interface		:= csp_case_main_safety_interface._SD10300_drv_ChA, 
			group						:= csp_case_main_safety_drives_SD10300.sig, 
			CONVERSION_this				:= SD10300_drv);
	END_IF
		
	IF 	SD10300_drv.channel_B.has_channel
	THEN	
		soe_drive_enable_fsoe(
			handler						:= BOSCH_DRIVE_CHANNEL_B, 
			incoherence_timeout			:= INCOHERENCE_TIMEOUT_MS, 
			connection_interface		:= csp_case_main_safety_interface._SD10300_drv_ChB, 
			group						:= csp_case_main_safety_drives_SD10300.sig, 
			CONVERSION_this				:= SD10300_drv);
	END_IF
	
	(* SD10400 *)
	soe_drive_double_channel_init(
		object_name					:= CONCAT(prc_path, '_SD10400_drv'), 
		device_name					:= 'SD10400', 
		vendor						:= DRIVE_BOSCH_REXROTH, 
		standalone					:= FALSE, 
		channel_a_name				:= 'csp_case_fc_ls_lower_spreader_axis', 
		channel_b_name				:= 'csp_case_fc_ls_lower_follower_axis', 
		ethercat_master				:= csp_main.cabinet_ethercat_master, 
		process						:= prc, 
		CONVERSION_this				:= SD10400_drv);	
		
	soe_drive_add_power_supply(
		power_supply				:= PS2000_ps, 
		CONVERSION_this				:= SD10400_drv);
		
	IF 	SD10400_drv.channel_a.has_channel
	THEN	
		soe_drive_enable_fsoe(
			handler						:= BOSCH_DRIVE_CHANNEL_A, 
			incoherence_timeout			:= INCOHERENCE_TIMEOUT_MS, 
			connection_interface		:= csp_case_main_safety_interface._SD10400_drv_ChA, 
			group						:= csp_case_main_safety_drives_SD10400.sig, 
			CONVERSION_this				:= SD10400_drv);
	END_IF
		
	IF 	SD10400_drv.channel_B.has_channel
	THEN	
		soe_drive_enable_fsoe(
			handler						:= BOSCH_DRIVE_CHANNEL_B, 
			incoherence_timeout			:= INCOHERENCE_TIMEOUT_MS, 
			connection_interface		:= csp_case_main_safety_interface._SD10400_drv_ChB, 
			group						:= csp_case_main_safety_drives_SD10400.sig, 
			CONVERSION_this				:= SD10400_drv);
	END_IF
	
	(* SD11000 *)
	soe_drive_double_channel_init(
		object_name					:= CONCAT(prc_path, '_SD11000_drv'), 
		device_name					:= 'SD11000', 
		vendor						:= DRIVE_BOSCH_REXROTH, 
		standalone					:= FALSE, 
		channel_a_name				:= 'csp_case_discharge_reject_belt_axis', 
		channel_b_name				:= '', 
		ethercat_master				:= csp_main.cabinet_ethercat_master, 
		process						:= prc, 
		CONVERSION_this				:= SD11000_drv);	
		
	soe_drive_add_power_supply(
		power_supply				:= PS2000_ps, 
		CONVERSION_this				:= SD11000_drv);
		
	IF 	SD11000_drv.channel_a.has_channel
	THEN	
		soe_drive_enable_fsoe(
			handler						:= BOSCH_DRIVE_CHANNEL_A, 
			incoherence_timeout			:= INCOHERENCE_TIMEOUT_MS, 
			connection_interface		:= csp_case_main_safety_interface._SD11000_drv_ChA, 
			group						:= csp_case_main_safety_drives_SD11000.sig, 
			CONVERSION_this				:= SD11000_drv);
	END_IF
		
	IF 	SD11000_drv.channel_B.has_channel
	THEN	
		soe_drive_enable_fsoe(
			handler						:= BOSCH_DRIVE_CHANNEL_B, 
			incoherence_timeout			:= INCOHERENCE_TIMEOUT_MS, 
			connection_interface		:= csp_case_main_safety_interface._SD11000_drv_ChB, 
			group						:= csp_case_main_safety_drives_SD11000.sig, 
			CONVERSION_this				:= SD11000_drv);
	END_IF
	
	(* SD15000 *)
	soe_drive_double_channel_init(
		object_name					:= CONCAT(prc_path, '_SD15000_drv'), 
		device_name					:= 'SD15000', 
		vendor						:= DRIVE_BOSCH_REXROTH, 
		standalone					:= FALSE, 
		channel_a_name				:= '', 
		channel_b_name				:= '', 
		ethercat_master				:= csp_main.cabinet_ethercat_master, 
		process						:= prc, 
		CONVERSION_this				:= SD15000_drv);	
		
	soe_drive_add_power_supply(
		power_supply				:= PS2000_ps, 
		CONVERSION_this				:= SD15000_drv);
		
	IF 	SD15000_drv.channel_a.has_channel
	THEN	
		soe_drive_enable_fsoe(
			handler						:= BOSCH_DRIVE_CHANNEL_A, 
			incoherence_timeout			:= INCOHERENCE_TIMEOUT_MS, 
			connection_interface		:= csp_case_main_safety_interface._SD15000_drv_ChA, 
			group						:= csp_case_main_safety_drives_SD15000.sig, 
			CONVERSION_this				:= SD15000_drv);
	END_IF
		
	IF 	SD15000_drv.channel_B.has_channel
	THEN	
		soe_drive_enable_fsoe(
			handler						:= BOSCH_DRIVE_CHANNEL_B, 
			incoherence_timeout			:= INCOHERENCE_TIMEOUT_MS, 
			connection_interface		:= csp_case_main_safety_interface._SD15000_drv_ChB, 
			group						:= csp_case_main_safety_drives_SD15000.sig, 
			CONVERSION_this				:= SD15000_drv);
	END_IF
	
	(* SD26000 *)
	soe_drive_double_channel_init(
		object_name					:= CONCAT(prc_path, '_SD26000_drv'), 
		device_name					:= 'SD26000', 
		vendor						:= DRIVE_BOSCH_REXROTH, 
		standalone					:= FALSE, 
		channel_a_name				:= 'csp_case_tr_squaring_os_leading_axis', 
		channel_b_name				:= 'csp_case_tr_squaring_os_trailing_axis', 
		ethercat_master				:= csp_main.cabinet_ethercat_master, 
		process						:= prc, 
		CONVERSION_this				:= SD26000_drv);	
		
	soe_drive_add_power_supply(
		power_supply				:= PS2000_ps, 
		CONVERSION_this				:= SD26000_drv);
		
	IF 	SD26000_drv.channel_a.has_channel
	THEN	
		soe_drive_enable_fsoe(
			handler						:= BOSCH_DRIVE_CHANNEL_A, 
			incoherence_timeout			:= INCOHERENCE_TIMEOUT_MS, 
			connection_interface		:= csp_case_main_safety_interface._SD26000_drv_ChA, 
			group						:= csp_case_main_safety_drives_SD26000.sig, 
			CONVERSION_this				:= SD26000_drv);
	END_IF
		
	IF 	SD26000_drv.channel_B.has_channel
	THEN	
		soe_drive_enable_fsoe(
			handler						:= BOSCH_DRIVE_CHANNEL_B, 
			incoherence_timeout			:= INCOHERENCE_TIMEOUT_MS, 
			connection_interface		:= csp_case_main_safety_interface._SD26000_drv_ChB, 
			group						:= csp_case_main_safety_drives_SD26000.sig, 
			CONVERSION_this				:= SD26000_drv);
	END_IF
	
	(* SD26100 *)
	soe_drive_double_channel_init(
		object_name					:= CONCAT(prc_path, '_SD26100_drv'), 
		device_name					:= 'SD26100', 
		vendor						:= DRIVE_BOSCH_REXROTH, 
		standalone					:= FALSE, 
		channel_a_name				:= 'csp_case_tr_squaring_ls_leading_axis', 
		channel_b_name				:= 'csp_case_tr_squaring_ls_trailing_axis', 
		ethercat_master				:= csp_main.cabinet_ethercat_master, 
		process						:= prc, 
		CONVERSION_this				:= SD26100_drv);	
		
	soe_drive_add_power_supply(
		power_supply				:= PS2000_ps, 
		CONVERSION_this				:= SD26100_drv);
		
	IF 	SD26100_drv.channel_a.has_channel
	THEN	
		soe_drive_enable_fsoe(
			handler						:= BOSCH_DRIVE_CHANNEL_A, 
			incoherence_timeout			:= INCOHERENCE_TIMEOUT_MS, 
			connection_interface		:= csp_case_main_safety_interface._SD26100_drv_ChA, 
			group						:= csp_case_main_safety_drives_SD26100.sig, 
			CONVERSION_this				:= SD26100_drv);
	END_IF
		
	IF 	SD26100_drv.channel_B.has_channel
	THEN	
		soe_drive_enable_fsoe(
			handler						:= BOSCH_DRIVE_CHANNEL_B, 
			incoherence_timeout			:= INCOHERENCE_TIMEOUT_MS, 
			connection_interface		:= csp_case_main_safety_interface._SD26100_drv_ChB, 
			group						:= csp_case_main_safety_drives_SD26100.sig, 
			CONVERSION_this				:= SD26100_drv);
	END_IF
	
END_IF

IF objects_running()
THEN
	process_cycle(prc);
	
	power_supply_cycle(PS2000_ps);
	
	soe_drive_cycle(SD2100_drv);
	soe_drive_cycle(SD2200_drv);
	soe_drive_cycle(SD2300_drv);
	soe_drive_cycle(SD2400_drv);
	soe_drive_cycle(SD2500_drv);
	soe_drive_cycle(SD12000_drv);
	soe_drive_cycle(SD8000_drv);
	soe_drive_cycle(SD8100_drv);
	soe_drive_cycle(SD8200_drv);
	soe_drive_cycle(SD8300_drv);
	soe_drive_cycle(SD8400_drv);
	soe_drive_cycle(SD8500_drv);
	soe_drive_cycle(SD8600_drv);
	soe_drive_cycle(SD10000_drv);
	soe_drive_cycle(SD10100_drv);
	soe_drive_cycle(SD10200_drv);
	soe_drive_cycle(SD10300_drv);
	soe_drive_cycle(SD10400_drv);
	soe_drive_cycle(SD11000_drv);
	soe_drive_cycle(SD15000_drv);
	soe_drive_cycle(SD26000_drv);
	soe_drive_cycle(SD26100_drv);

END_IF
END_ACTION

ACTION _read_process_image:
;
END_ACTION

ACTION _read_var_input:
;
END_ACTION

ACTION _set_runtime_properties:
;
END_ACTION

ACTION _write_output:
;
END_ACTION

END_PROGRAM

// ---- Application/CSP/Case/Main/csp_case_main.TcPOU
(*********************************** G.D S.p.A. - Technical Department ***********************************
============= PROGRAM INFO ============
FOLDER:             TBD
MACHINES INVOLVED:  TBD 

============= DESCRIPTION =============
csp main program

============= REVISIONS ===============
Date		Version	 	Author      	Description             
----------	-------		------------  	--------------------------------------------
2019/04/05 	0000.00	 	M.Grasso		Creation of the PRG

**********************************************************************************************************)
(*$R
	process_ref := prc;
$*)
PROGRAM csp_case_main
VAR
	prc:												process;
	prc_path:											STRING;
END_VAR


VAR_OUTPUT
	o_reset_button:										BOOL;
	o_start_button:										BOOL;
END_VAR

_read_var_input();

_object_manager();

IF NOT objects_running()
THEN
	RETURN;	
END_IF

_read_process_image();

_mode_manager();

CASE process_get_mode(prc) of
	MODE_ABSENT,
	MODE_INACTIVE:
		RETURN;
	MODE_TEST:
		_handle_process_test();
END_CASE

_set_runtime_properties();

(********************************* BODY *********************************)

(************************************************************************)

_handle_messages();

_write_output();

ACTION _handle_messages:
;
END_ACTION

ACTION _handle_process_test:
;
END_ACTION

ACTION _mode_manager:
IF process_mode_req_is_pending(prc)
THEN
    process_apply_mode_req_first_step(prc);
    CASE process_get_mode(prc) OF
        MODE_TO_ABSENT:
			;
        MODE_TO_INACTIVE:
			;
        MODE_TO_TEST:
			;
        MODE_TO_OPERATIONAL:
			;
    END_CASE
    process_apply_mode_req_second_step(prc);
END_IF
END_ACTION

ACTION _object_manager:
IF objects_initialization()
THEN
	sub_process_init(
		object_name					:= 'csp_case_main.prc', 
		process						:= csp_case.prc, 
		CONVERSION_this				:= prc);
		
	prc_path 						:= process_get_path(prc);
END_IF

IF objects_running()
THEN
	process_cycle(prc);
END_IF
END_ACTION

ACTION _read_process_image:
;
END_ACTION

ACTION _read_var_input:

END_ACTION

ACTION _set_runtime_properties:
;
END_ACTION

ACTION _write_output:
o_reset_button	:= csp_case_main_services_pushbuttons.reset_pressed;
o_start_button	:= csp_case_main_services_pushbuttons.start_pressed;
END_ACTION

END_PROGRAM

// ---- Application/CSP/Main/Interface/csp_main_interface.TcPOU
(*********************************** G.D S.p.A. - Technical Department ***********************************
============= PROGRAM INFO ============
FOLDER:             TBD
MACHINES INVOLVED:  TBD 

============= DESCRIPTION =============
csp main interface program

============= REVISIONS ===============
Date		Version	 	Author      	Description             
----------	-------		------------  	--------------------------------------------
2019/09/27 	0000.00	 	M.Grasso		Creation of the PRG

**********************************************************************************************************)
(*$R
	process_ref := prc;
$*)
PROGRAM csp_main_interface
VAR
	prc:								process;
	prc_path:							STRING;
	
	alarm_state:						csp_main_interface_csv_read;
	alarm_state_next:					csp_main_interface_csv_read;
	
	
	debug_state_machine:				BOOL;
	debug_state_machine_one_step:		BOOL;
	
	
	first_stop_object_name:				STRING := '';
	first_stop_object_name_short:		STRING := '';
	
	machine_fault_cleared_r_trig:		R_TRIG;
	
	new_alarm_rising:					BOOL;
	new_alarm:							BOOL;
	
	alarm_list_filename:				T_MaxString := 'C:\Casepacker_fault_list.csv';
	
	timeout:							TIME := T#5S;
	
	file_opened:						BOOL;
	
	fb_open:							FB_FileOpen;
	fb_read:							FB_FileGets;
	fb_close:							FB_FileClose;
	
	test_open:							BOOL;
	test_read:							BOOL;
	test_close:							BOOL;
	
	object_name:						T_MaxString;
	new_line_count:						INT;
	
	stop_object:						ARRAY[0..2] OF T_MaxString;
	sSeparator:							STRING(1) := ',';
	i:									INT := 0;
	char_count:							INT;
	
	alarm_found:						BOOL := FALSE;
	alarm_id_string:					STRING;
	alarm_id:							INT;
	
	alarm_match_length:					INT;
	
	eof:								BOOL;
	
	stop_0_lower:						T_MaxString;
	first_stop_lower:					T_MaxString;
	
	int_test:							INT;
	alarm_ID_from_python:				DINT;
	
	python_alive:						BOOL;
	python_alive_flt:					filter;
	python_parse_running:				BOOL := FALSE;
	
	Cartoner_Communication_OK:			BOOL;
	Cartoner_Faulted:					BOOL;
	Cartoner_Running:					BOOL;
	Cartoner_StopRequest:				BOOL;
	Cartoner_RunOutRequest:				BOOL;
	Cartoner_Estop:						BOOL;
	Cartoner_Stop_Request_aem:			message;
	cartoner_stop_request_delay_tmr:	timer;
	cartoner_stop_request_delay:		DINT:= 3000;
	cartoner_stop_bypass_request:		BOOL:= FALSE;
	communication_time_out_tmr:			timer;
	communication_failure_nsm:			message;
	first_scan:							BOOL;
	open_error_reset_delay: 			TON;
	open_error_reset: 					BOOL;
	open_error_PT: 						TIME := T#5S;
	open_error_done: 					BOOL;
	
	downstream_hold_motcond:			motorization_conditioner;
END_VAR

_read_var_input();

_object_manager();

IF NOT objects_running()
THEN
	first_scan:= TRUE;
	timer_restart(1000,	communication_time_out_tmr);
	RETURN;	
END_IF

_read_process_image();

_mode_manager();

CASE process_get_mode(prc) OF
	MODE_ABSENT,
	MODE_INACTIVE:
		RETURN;
	MODE_TEST:
		_handle_process_test();
END_CASE

_set_runtime_properties();

(********************************* BODY *********************************)

(* Alive bit *)
IF	Cartoner_Communication_OK = RAJ_To_Cartoner[0].0
	OR
	first_scan
THEN
	timer_restart(1000,	communication_time_out_tmr);
END_IF

RAJ_To_Cartoner[0].0	:= NOT Cartoner_Communication_OK;

IF	timer_is_expired(communication_time_out_tmr)
THEN
	process_message_set(1, 0, 0, communication_failure_nsm);
ELSE
	process_message_reset(communication_failure_nsm);
END_IF



//BJS -- Cartoner Communication
//RAJ_To_Cartoner[0].0		:= TRUE;
RAJ_To_Cartoner[0].1 		:= NOT machine_is_running(csp.mch) (*AND NOT axis_is_moving(csp_main_motorization_virtualManager.axis) AND NOT message_is_on(csp_case_discharge_reject_sensors.downstream_backup_di_dchk.alarm_asm.message) AND NOT message_is_on(csp_main_interface.Cartoner_Stop_Request_aem)*);
RAJ_To_Cartoner[0].2 		:= machine_is_running(csp.mch);
RAJ_To_Cartoner[0].3 		:= axis_is_moving(csp_transfer_infeed_metering_belt.axis) AND csp_transfer_infeed_metering_belt.ok_to_start_temp_infeed_belt AND csp_transfer_infeed.run_infeed_belts_orginal;//NAW added 4_19_23
RAJ_To_Cartoner[0].4 		:= digital_output_is_active(csp_case_discharge_reject_modsort.MODSORT_FWD_RUN_do);
RAJ_To_Cartoner[0].5 		:= message_is_on(csp_case_discharge_reject_sensors.downstream_backup_di_dchk.alarm_asm.message) OR message_is_on(csp_main_interface.Cartoner_Stop_Request_aem); // machine is held
RAJ_To_Cartoner[0].31		:= csp_main.i_csp_data_ref^.Status.RunOutComplete;
RAJ_To_Cartoner[19]			:= REAL_TO_DINT(machine_get_nominal_velocity(csp.mch));

Cartoner_Communication_OK	:= Cartoner_To_RAJ[0].0;
Cartoner_Faulted 			:= Cartoner_To_RAJ[0].1;
Cartoner_Running			:= Cartoner_To_RAJ[0].2;
Cartoner_StopRequest		:= Cartoner_To_RAJ[0].3;
Cartoner_Estop				:= Cartoner_To_RAJ[0].4;
Cartoner_RunOutRequest		:= Cartoner_To_RAJ[0].31;

(*
IF csp.o_machine_is_stopped OR ( NOT(csp_main_motorization_manager.suspend_conditions) AND timer_is_expired(cartoner_stop_request_delay_tmr))
	THEN
		process_message_reset(Cartoner_Stop_Request_aem);
END_IF
*)
IF 	Cartoner_StopRequest 
	AND NOT cartoner_stop_bypass_request
	AND NOT csp_case_main_services.dry_cycle_mode
	AND NOT message_is_on(csp_main_jogmanager.jog_is_active_wem)
THEN
	process_message_set(1, 1, 1, Cartoner_Stop_Request_aem);
	
	IF	csp_main_motorization_manager.debug_Enable_new_conditioners (* Selector on HMI while still being tested *)
	THEN
		motorization_conditioner_hold(downstream_hold_motcond);
		motorization_conditioner_velocity_limit_activate(downstream_hold_motcond);
	END_IF
ELSE
	process_message_reset(Cartoner_Stop_Request_aem);
	motorization_conditioner_unhold(downstream_hold_motcond);
	motorization_conditioner_velocity_limit_deactivate(downstream_hold_motcond);
END_IF

(* SETS PYTHON ALIVE BACK TO FALSE TO ALLOW FOR PYTHON CODE TO CHANGE AGAIN *)
IF 	python_alive
	AND filter_is_on(python_alive_flt)
THEN
	python_alive := FALSE;
END_IF

(* CHANGES TO PARSE BY PYTHON *)
IF 	filter_is_on(python_alive_flt)
	AND alarm_state <= 10
THEN
	python_parse_running := TRUE;
END_IF

(* CHANGES TO LOCAL PARSE *)
IF 	filter_is_off(python_alive_flt)
	AND alarm_state <= 10
THEN
	python_parse_running := FALSE;
END_IF

(* Resets Identified Alarm ID after machine has been reset or started *)
IF 	machine_is_ready(csp.mch)
	OR
	machine_is_running(csp.mch)
	AND NOT motorization_manager_is_holding(csp_main_motorization_manager.motm) 
	AND NOT motorization_manager_is_held(csp_main_motorization_manager.motm) 
THEN
	alarm_id := 0;
END_IF

(* SORTS BETWEEN PYTHON PARSE AND LOCAL PARSE *)
IF 	python_parse_running
THEN
		;
(* LOCAL PARSE CODE *)
ELSE
	
	machine_fault_cleared_r_trig(CLK := machine_is_ready(csp.mch));
	
	IF 	machine_fault_cleared_r_trig.Q
		AND alarm_state > 10
	THEN
		alarm_state_next := 200;
	END_IF
	
	
	CASE alarm_state OF
		
		0: // csv_read_idle
			IF 	machine_is_ready(csp.mch)
				OR machine_is_running(csp.mch)
			THEN
				first_stop_object_name := '';
				alarm_id := 0;
				alarm_state_next := 10;
			END_IF
			
			
		10: // csv_read_wait_for_alarm
			IF 	machine_is_stopped(csp.mch)
				OR machine_is_stop_emergency_active(csp.mch)
			THEN
				first_stop_object_name := csp.mch.first_stop_message^.object_name;
				alarm_state_next := 20;
			END_IF
	
			IF machine_is_running(csp.mch) 
				AND	csp_main_motorization_manager.Upstream_Wait
			THEN	
				alarm_id := (900);
			END_IF
			IF machine_is_running(csp.mch) 
			   AND	csp_main_motorization_manager.Downstream_Wait
			THEN	
				alarm_id := (901);
			END_IF
				
			IF machine_is_running(csp.mch) 
			   AND	downstream_hold_motcond.is_active
			   AND NOT machine_is_execute(csp.mch)
			THEN	
				alarm_id := (902);
			END_IF
			
		20: // csv_read_clear_variables
			alarm_found := FALSE;
			object_name := '';
			alarm_id := 0;
			stop_object[0] := '';
			stop_object[1] := '';
			stop_object[2] := '';
			eof := FALSE;
			first_stop_object_name_short := '';
			alarm_state_next := 30;
			
		30: // csv_read_trim_object_name
			first_stop_object_name_short := LEFT(first_stop_object_name, FIND(first_stop_object_name, '/') - 1);
		
			IF 	FIND(first_stop_object_name_short, '._') > 0
			THEN
				first_stop_object_name_short := REPLACE(first_stop_object_name_short, '.', 2, FIND(first_stop_object_name_short, '._'));
			END_IF
			
			alarm_state_next := 40;
			
		40: // csv_read_open_csv_file
			test_open := TRUE;
			
			IF 	fb_open.bBusy
			THEN
				alarm_state_next := 50;
			END_IF
			
		50: // csv_read_verify_open
			IF 	NOT fb_open.bError
			THEN
				test_open := FALSE;
				alarm_state_next := 60;
			ELSE
				;
			END_IF
			
		60: // csv_read_read_csv_file // WILL LOOP HERE TO ITERATE
			test_read := TRUE;
			
			IF 	fb_read.bBusy
				//OR
				//fb_read.bExecute
			THEN
				alarm_state_next := 70;
			END_IF
			
		70: // csv_read_verify_read
			IF 	NOT fb_read.bError
			THEN
				test_read := FALSE;
			
				object_name := '';
				
				stop_object[0] := '';
				stop_object[1] := '';
				stop_object[2] := '';
				
				alarm_state_next := 80;
			ELSE
				;
			END_IF
			
		80: // csv_read_parse_csv_stop_data
			IF object_name = ''
			THEN
				i := 0;
				object_name := CONCAT(fb_read.sLine, ','); // ADDS COMMA FOR EASY PARSING
			END_IF
			
			IF FIND(object_name, '._') > 0
			THEN
				REPLACE(object_name, '.', 2, FIND(object_name, '._')); // ELIMINATES ._ THAT IS IN SOME OBJECT NAMES
			END_IF
			
			IF stop_object[0] = ''
			THEN
				stop_object[0] := LEFT(object_name, FIND(object_name, sSeparator) - 1);
				object_name := DELETE(object_name, FIND(object_name, sSeparator) + 1, 0);
			END_IF
			
			IF 	stop_object[0] <> ''
				AND stop_object[1] = ''
			THEN
				stop_object[1] := LEFT(object_name, FIND(object_name, sSeparator) - 1);
				object_name := DELETE(object_name, FIND(object_name, sSeparator) + 1, 0);
			END_IF
			
			IF 	stop_object[0] <> ''
				AND stop_object[1] <> ''
				AND stop_object[2] = ''
			THEN
				stop_object[2] := LEFT(object_name, FIND(object_name, sSeparator) - 2);
			END_IF
			
			
			IF 	LEFT(stop_object[0], 1) <> '.'
			THEN
					;//stop_object[0] := CONCAT('.', stop_object[0]);
			END_IF
			
			IF stop_object[0] <> ''
				//AND LEFT(stop_object[0], 1) = '.'
				AND stop_object[1] <> ''
				AND stop_object[2] <> ''
			THEN
				//stop_object[2] := LEFT(stop_object[2], LEN(stop_object[2]) - 2);
				alarm_state_next := 90;
			END_IF
			
			
		90: // csv_read_compare_stop
			stop_0_lower := F_ToLCase(stop_object[0]);
			first_stop_lower := F_ToLCase(first_stop_object_name_short);
			
			IF 	FIND(stop_0_lower, first_stop_lower) > 0
			THEN
				alarm_state_next := 100;
			ELSE
				alarm_state_next := 60;
			END_IF
			
		100: // csv_read_alarm_found
			alarm_id_string := stop_object[2];
			alarm_id := STRING_TO_INT(alarm_id_string);
			
			alarm_found := TRUE;
			
			alarm_state_next := 200;
			
			
		200: // csv_read_close_csv_file
			test_close := TRUE;
			
			IF 	fb_close.bBusy
			THEN
				alarm_state_next := 210;
			END_IF
			
		210: // csv_read_close_csv_file_verify
			IF 	NOT fb_close.bError
			THEN
				test_close := FALSE;
					
				alarm_state_next := 0;
			END_IF
	
	END_CASE
	
	
	IF 	NOT debug_state_machine
		OR
		debug_state_machine_one_step
	THEN
		alarm_state := alarm_state_next;
		debug_state_machine_one_step := FALSE;
	END_IF
	

END_IF



(* Function blocks handle opening, reading, and closing the csv file to obtain alarm ID*)
fb_open(
	sNetId		:= '',
	sPathName	:= alarm_list_filename,
	nMode		:= FOPEN_MODEREAD,
	ePath		:= ,
	bExecute	:= test_open,
	tTimeout	:= timeout);

	
fb_close(
	sNetId		:= '',
	hFile		:= fb_open.hFile,
	bExecute	:= test_close,
	tTimeout	:= timeout);

fb_read(
	sNetId		:= '',
	hFile		:= fb_open.hFile,
	bExecute	:= test_read,
	tTimeout	:= timeout);

IF fb_close.bError
THEN
	test_close := FALSE;
	alarm_state_next := 0;
END_IF

IF fb_open.bError
THEN
	test_open := FALSE;
	alarm_state_next := 0;
END_IF

IF fb_read.bError
THEN
	test_read := FALSE;
	alarm_state_next := 0;
END_IF

(************************************************************************)

_handle_messages();

_write_output();

ACTION _handle_messages:
;
END_ACTION

ACTION _handle_process_test:
;
END_ACTION

ACTION _mode_manager:
IF process_mode_req_is_pending(prc)
THEN
    process_apply_mode_req_first_step(prc);
    CASE process_get_mode(prc) OF
        MODE_TO_ABSENT:
			;
        MODE_TO_INACTIVE:
			;
        MODE_TO_TEST:
			;
        MODE_TO_OPERATIONAL:
			;
    END_CASE
    process_apply_mode_req_second_step(prc);
END_IF
END_ACTION

ACTION _object_manager:
IF objects_initialization()
THEN
	sub_process_init(
		object_name					:= 'csp_main_interface.prc', 
		process						:= csp_main.prc, 
		CONVERSION_this				:= prc);
		
	prc_path 						:= process_get_path(prc);
	
	filter_init(
		object_name					:= CONCAT(prc_path, '_python_alive_flt'), 
		delay_off_on				:= 2000,
		delay_on_off				:= 2000,
		process						:= csp_main.prc, 
		CONVERSION_this				:= python_alive_flt);
		
		
	process_message_init(
		object_name:= CONCAT(prc_path, '_Cartoner_Stop_Request_aem'),
		behaviour:= MESSAGE_BEHAVIOUR_STATE,
		reset_timeout:= 0,
		disableable:= FALSE,
		individual_reset:= FALSE,
		machine_reaction:= MACHINE_REACTION_NO_STOP,
		typology:= MESSAGE_TYPOLOGY_OBLIGATION,
		process:= prc,
		CONVERSION_this:= Cartoner_Stop_Request_aem);
	
	timer_init(
		object_name					:=	CONCAT(prc_path, '_communication_time_out_tmr'),
		process						:=	prc,
		CONVERSION_this				:=	communication_time_out_tmr);
	
	process_message_init(
		object_name					:=	CONCAT(prc_path, '_communication_failure_nsm'),
		behaviour					:=	MESSAGE_BEHAVIOUR_STATE,
		reset_timeout				:=	0,
		disableable					:=	TRUE,
		individual_reset			:=	FALSE,
		machine_reaction			:=	MACHINE_REACTION_NO_STOP,
		typology					:=	MESSAGE_TYPOLOGY_NORMAL,
		process						:=	prc,
		CONVERSION_this				:=	communication_failure_nsm);
		
	timer_init(
		object_name					:=	CONCAT(prc_path, '_cartoner_stop_request_delay_tmr'),
		process						:=	prc,
		CONVERSION_this				:=	cartoner_stop_request_delay_tmr);
	
	motorization_conditioner_init(
		object_name := CONCAT(prc_path, '_downstream_hold_motcond'),
		velocity_limit := 0,
		velocity_limit_active := FALSE,
		idle_handshake_active := FALSE,
		execute_handshake_active := FALSE,
		hold_handshake_active := FALSE,
		suspend_handshake_active := FALSE,
		complete_handshake_active := FALSE,
		abort_handshake_active := FALSE,
		stop_handshake_active := FALSE,
		origin := MOTORIZATION_CONDITIONER_ORIGIN_EXTERNAL_DOWN,
		manager := csp_main_motorization_manager.motm,
		process := prc,
		CONVERSION_this := downstream_hold_motcond);
	
END_IF

IF objects_running()
THEN
	process_cycle(prc);
	motorization_conditioner_cycle(downstream_hold_motcond);

	filter_cycle(python_alive, python_alive_flt);
END_IF
END_ACTION

ACTION _read_process_image:
;
END_ACTION

ACTION _read_var_input:
;
END_ACTION

ACTION _set_runtime_properties:
;
END_ACTION

ACTION _write_output:
;
END_ACTION

END_PROGRAM

// ---- Application/CSP/Transfer/Infeed/csp_transfer_infeed.TcPOU
(*********************************** G.D S.p.A. - Technical Department ***********************************
============= PROGRAM INFO ============
FOLDER:             TBD
MACHINES INVOLVED:  TBD 

============= DESCRIPTION =============
csp machine declaration

============= REVISIONS ===============
Date		Version	 	Author      	Description             
----------	-------		------------  	--------------------------------------------
2019/04/05 	0000.00	 	M.Grasso		Creation of the PRG

**********************************************************************************************************)
(*$R process_ref := prc; $*)
PROGRAM csp_transfer_infeed
VAR
	
	prc:											process;
	prc_path:										STRING;
	
	temp_belt_run AT %Q*:							BOOL;
	
	run_infeed_belts:								BOOL;
	
	belt_accumulation_fsm_status:					csp_transfer_infeed_belt_status_enum;	(*$M desc := Conveyor Belt Accumulation FSM Status; $*)
	belt_metering_fsm_status:						csp_transfer_infeed_belt_status_enum;	(*$M desc := Conveyor Belt Metering Status; $*)
	belt_waterfall_fsm_status:						csp_transfer_infeed_belt_status_enum;	(*$M desc := Conveyor Belt Waterfall Status; $*)
	
	run_do:											digital_output;
	
	csp_running_velocity_PPM:						LREAL;	(*$M unit :=  PPM; desc := Cartoner Running Velocity; $*)
	csp_running_velocity_mmpm:						LREAL;	(*$M unit :=  mm/s; desc := CasePacker Running Velocity; $*)
	velocity_req_perc:								REAL:=0.0;	(*$M unit := %; desc := Pump Speed Request Output ; $*)
	velocity_req_limited_perc:						REAL:=0.0;	(*$M unit := %; desc := Pump Speed Limited Output ; $*)
	velocity_req_limited_old_perc:					REAL;
	
	metering_running_velocity_mmpm:					LREAL;
	waterfall_accum_running_velocity_mmpm:			LREAL;
	
	
	debug_conveyor:									BOOL;		
	manual_velocity_ppm_override:					BOOL;
	manual_velocity_ppm:							LREAL := 15;
	
	metering_belt_rpm_per_mm:						LREAL := 0.0062;
	metering_belt_hz_per_rpm:						LREAL := 0.1739;
	metering_belt_rpm_req:							LREAL;
	metering_belt_hz_req:							LREAL;
	
	metering_belt_hz_per_mm:						LREAL := 0.0000663349917; (* 1Hz = 15075 mm/min *)
	
	waterfall_belt_rpm_per_mm:						LREAL := 0.0062;
	waterfall_belt_hz_per_rpm:						LREAL := 0.1739;
	waterfall_belt_rpm_req:							LREAL;
	waterfall_belt_hz_req:							LREAL;
	
	waterfall_belt_hz_per_mm:						LREAL := 0.00006557377; (* 1Hz = 15250 mm/min *)
	
	accumulation_belt_rpm_per_mm:					LREAL := 0.0020595; (* 173RPM = 84 m/min - NEEDS TO CHANGE*)
	accumulation_belt_hz_per_rpm:					LREAL := 0.3468; (* 173RPM = 60Hz *)
	accumulation_belt_rpm_req:						LREAL;
	accumulation_belt_hz_req:						LREAL;
	
	accumulation_belt_hz_per_mm:					LREAL := 0.00002160994; (* 1Hz = 46275 mm/min *)
	
	rm_cartoner_speed:								LREAL := 60;
	
	
	belts_time_out_tmr:								timer;
	belts_faulted_aem:	 							message;
	infeed_belts_surge_percent:						LREAL := 30;
	
	stop_signal_delay: 								Ton;
	delay_stop_signal: 								BOOL;
	run_infeed_belts_orginal: 						BOOL;
END_VAR

VAR_INPUT

	i_downstream_ready:								BOOL;					(*$M desc := Downstream Process Ready; $*)
	i_upstream_running:								BOOL;
	i_upstream_immediate_stop:						BOOL;
	i_upstream_velocity:							LREAL;

END_VAR

VAR CONSTANT
	MIN_VELOCITY_PERC:								REAL := 10;
	MAX_VELOCITY_PERC:								REAL := 100;
	MAX_VELOCITY_MMPS:								REAL := 1500;
	MIN_MACHINE_SPEED_FOR_BELTS:					INT := 10;
END_VAR

_read_var_input();

_object_manager();

IF NOT objects_running()
THEN
	RETURN;	
END_IF

_read_process_image();

_mode_manager();

CASE process_get_mode(prc) OF
	MODE_ABSENT,
	MODE_INACTIVE:
		RETURN;
	MODE_TEST:
		_handle_process_test();
END_CASE


_set_runtime_properties();

(********************************* BODY *********************************)
(************************************************************************)


IF axis_is_moving(csp_transfer_infeed_metering_belt.axis)
	OR
	axis_is_moving(csp_transfer_infeed_waterfall_belt.axis)
	AND NOT csp_transfer_infeed_accumulation_level.stop_upstream_belts
THEN
	temp_belt_run := TRUE;
ELSE
	temp_belt_run := FALSE;
END_IF



IF	machine_is_running(csp.mch)
	AND csp_main_motorization_manager.motm.actual_velocity > 0
THEN
	IF	timer_is_expired(belts_time_out_tmr)
		AND csp_transfer_infeed_metering_belt.fsm_status <> CSP_TRANSFER_INFEED_BELT_STATUS_RUNNING
		AND csp_transfer_infeed_waterfall_belt.fsm_status <> CSP_TRANSFER_INFEED_WATERFALL_BELT_STATUS_RUNNING
		AND csp_transfer_infeed_accumulation_belt.fsm_status <> CSP_TRANSFER_INFEED_ACCUMULATION_BELT_STATUS_RUNNING
	THEN
		//process_message_set(1, 0, 0, belts_faulted_aem);
	END_IF
ELSE
	timer_restart(2500, belts_time_out_tmr);
END_IF


(* ENABLE CONDITION FOR ALL INFEED BELTS *)
run_infeed_belts :=
	(
		motorization_manager_is_execute(csp_main_motorization_manager.motm)
		OR
		motorization_manager_is_holding(csp_main_motorization_manager.motm)
		OR
		motorization_manager_is_held(csp_main_motorization_manager.motm)
		OR
		motorization_manager_is_unholding(csp_main_motorization_manager.motm)
		OR
		csp_main_motorization_virtualManager.axis.actual_velocity > 0 //catches suspend
		OR
		NOT delay_stop_signal 
	)
	AND
	process_is_ready(prc);

//Added to continue the infeed belts to run 2 seconds after a stop	
stop_signal_delay(IN:= csp_main_motorization_virtualManager.axis.actual_velocity < 1, PT:=T#2S , Q=> delay_stop_signal , ET=> );

run_infeed_belts_orginal :=
	(
		motorization_manager_is_execute(csp_main_motorization_manager.motm)
		OR
		motorization_manager_is_holding(csp_main_motorization_manager.motm)
		OR
		motorization_manager_is_held(csp_main_motorization_manager.motm)
		OR
		motorization_manager_is_unholding(csp_main_motorization_manager.motm)
		OR
		csp_main_motorization_virtualManager.axis.actual_velocity > 0 //catches suspend
	)
	AND
	process_is_ready(prc);
	
IF manual_velocity_ppm_override
THEN
	csp_running_velocity_PPM := manual_velocity_ppm;
ELSE
	csp_running_velocity_PPM := csp_main_brand.case_pattern.case_pattern_L * csp_main_brand.case_pattern.case_pattern_W * csp_main_brand.surge_case_rate_ppm;
END_IF

csp_running_velocity_mmpm := 	MAX(csp_main_motorization_manager.motm.actual_velocity_setpoint, MIN_MACHINE_SPEED_FOR_BELTS) 
								*
								csp_main_brand.case_pattern.case_pattern_L
								*
								csp_main_brand.case_pattern.case_pattern_W;
								

(* USED FOR METERING BELTS SINCE SOMETIMES IN DIFFERENT ORIENTATION *)								
metering_running_velocity_mmpm := 	csp_running_velocity_mmpm
									*
									(
										SEL(csp_main_brand.Rollover_Carton,
											csp_main_brand.carton_dimension.carton_size_L_mm, 
											csp_main_brand.carton_dimension.carton_size_W_mm) (* SELECTED IF ROLLOVER IS TRUE *)
										//csp_main_brand.carton_dimension.carton_size_W_mm
										+ 
										csp_main_brand.metering_carton_gap
									)
									*
									(
										(infeed_belts_surge_percent / 100) + 1
									);

(* USED FOR WATERFALL AND ACCUMULATION BELTS *)
waterfall_accum_running_velocity_mmpm :=	csp_running_velocity_mmpm
									*
									(
										SEL(csp_main_brand.Rollover_Carton,
											csp_main_brand.carton_dimension.carton_size_W_mm, 
											csp_main_brand.carton_dimension.carton_size_L_mm) (* SELECTED IF ROLLOVER IS TRUE *)
										+ 
										csp_main_brand.post_waterfall_carton_gap
									)
									*
									(
										(infeed_belts_surge_percent / 100) + 1
									);

							
(* Metering Belt Req Velocity *)	
metering_belt_rpm_req := 	metering_running_velocity_mmpm
							*
							metering_belt_rpm_per_mm
							*
							( 1 + (csp_transfer_infeed_metering_belt.override_percentage_par / 100)); (* mm per minute *)
							


(* Waterfall Belt Req Velocity *)	
waterfall_belt_rpm_req := 	waterfall_accum_running_velocity_mmpm 
							* 
							waterfall_belt_rpm_per_mm
							*
							( 1 + (csp_transfer_infeed_waterfall_belt.override_percentage_par / 100)); (* mm per minute *)


(* Accumulation Belt Req Velocity *)	
accumulation_belt_rpm_req :=	waterfall_accum_running_velocity_mmpm
								*
								accumulation_belt_rpm_per_mm
								*
								( 1 + (csp_transfer_infeed_accumulation_belt.override_percentage_par / 100)); (* mm per minute *)
							
									
velocity_req_perc := 	csp_running_velocity_mmpm
						/
						MAX_VELOCITY_MMPS
						*
						100
						;
						
IF	run_infeed_belts
	OR
	debug_conveyor
THEN
	velocity_req_limited_perc := MIN(velocity_req_perc,MAX_VELOCITY_PERC);
	velocity_req_limited_perc := MAX(velocity_req_limited_perc, MIN_VELOCITY_PERC);
ELSE
	velocity_req_limited_perc := 0;
END_IF									

(************************************************************************)
_handle_messages();

_write_output();

ACTION _handle_messages:
;
END_ACTION

ACTION _handle_process_test:
;
END_ACTION

ACTION _mode_manager:
IF process_mode_req_is_pending(prc)
THEN
    process_apply_mode_req_first_step(prc);
    CASE process_get_mode(prc) OF
        MODE_TO_ABSENT:
			;
        MODE_TO_INACTIVE:
			;
        MODE_TO_TEST:
			velocity_req_limited_perc := 0;
			velocity_req_perc := 0;
        MODE_TO_OPERATIONAL:
			;
    END_CASE
    process_apply_mode_req_second_step(prc);
END_IF
END_ACTION

ACTION _object_manager:
IF objects_initialization()
THEN
	sub_process_init(
		object_name					:= 'csp_transfer_infeed.prc', 
		process						:= csp_transfer.prc, 
		CONVERSION_this				:= prc);
		
	prc_path 						:= process_get_path(prc);
	
	digital_output_init(
		object_name				:= CONCAT(prc_path, '_run_do'),
		polarity_direct			:= TRUE,
		process					:= prc,
		CONVERSION_this					:= run_do);

		
	process_message_init(
		object_name					:=	CONCAT(prc_path, '_belts_faulted_aem'), 
		behaviour					:=	MESSAGE_BEHAVIOUR_EVENT,
		reset_timeout				:=	0,
		disableable					:=	TRUE,
		individual_reset			:=	FALSE,
		machine_reaction			:=	MACHINE_REACTION_NORMAL_STOP,
		typology					:=	MESSAGE_TYPOLOGY_ABNORMAL,
		process						:=	prc,
		CONVERSION_this				:=	belts_faulted_aem);
	
	timer_init(
		object_name					:= CONCAT(prc_path, '_belts_time_out_tmr'),
		process						:= prc,
		CONVERSION_this				:= belts_time_out_tmr);	
		

END_IF

IF objects_running()
THEN
	process_cycle(prc);	
END_IF
END_ACTION

ACTION _read_process_image:
;
END_ACTION

ACTION _read_var_input:
i_downstream_ready:= TRUE;

i_upstream_running:=	NOT machine_is_stopped(csp.mch)
						AND
						process_mode_is_operational(csp_main_motorization_manager.prc);
						
i_upstream_immediate_stop:= FALSE; (* To Be Changed - Marco*)
i_upstream_velocity:= csp_running_velocity_mmpm;
END_ACTION

ACTION _set_runtime_properties:
;
END_ACTION

ACTION _write_output:
;
END_ACTION

END_PROGRAM

// ---- Application/CSP/Main/Motorization/Snapshot/csp_main_motorization_set_snapshot.TcPOU
(*********************************** G.D S.p.A. - Technical Department ***********************************
============= PROGRAM INFO ============
FOLDER:             TBD
MACHINES INVOLVED:  TBD 

============= DESCRIPTION =============
csp main motorization manager snapshot set function

============= REVISIONS ===============
Date		Version	 	Author      	Description             
----------	-------		------------  	--------------------------------------------
2019/04/27 	0000.00	 	M.Grasso		Creation of the PRG

**********************************************************************************************************)

FUNCTION csp_main_motorization_set_snapshot : VOID
VAR_INPUT
    errorID_1:				DINT;			(* Field for specify the faults code or enter
								   				more message info *)
    errorID_2:				DINT;			(* Field for specify the faults code or enter
								   				more message info *)
    errorID_3:				DINT;			(* Field for specify the faults code or enter
								   				more message info *)
	reason:					STRING := '';
	connection_status:		INT;
END_VAR

VAR_IN_OUT
    CONVERSION_this:		csp_main_motorization_snapshot;
								(* wu_main_motorization_manager_snapshot snapshot reference *)
END_VAR

IF	message_set(
		errorID_1		:= errorID_1, 
		errorID_2		:= errorID_2, 
		errorID_3		:= errorID_3, 
		CONVERSION_this	:= CONVERSION_this.message)
THEN
	CONVERSION_this.reason 				:= reason;
	CONVERSION_this.connection_status	:= connection_status;
end_if

END_FUNCTION

// ---- Application/CSP/Main/Motorization/Snapshot/csp_main_motorization_init_snapshot.TcPOU
(*********************************** G.D S.p.A. - Technical Department ***********************************
============= PROGRAM INFO ============
FOLDER:             TBD
MACHINES INVOLVED:  TBD 

============= DESCRIPTION =============
csp main motorization manager snapshot init function

============= REVISIONS ===============
Date		Version	 	Author      	Description             
----------	-------		------------  	--------------------------------------------
2019/04/27 	0000.00	 	M.Grasso		Creation of the PRG

**********************************************************************************************************)

FUNCTION csp_main_motorization_init_snapshot : VOID
VAR_INPUT	
	message_name:			STRING(MAX_OBJ_NAME_LENGTH);
	behaviour:				message_behaviour_enum;			(* Message type. State or event *)
	reset_timeout:			UDINT;							(* Timeout of reset attempt valid for messages
															   with <a href="#message_behaviour_enum"><i>behaviour</i></a>
															   = MESSAGE_BEHAVIOUR_TRY_AND_CHECK *)
    disableable:        	BOOL;							(* Indicates the possibility
																to disable the message by HMI *)
    individual_reset:   	BOOL;							(* Need explicit reset by
																HMI for acknowlege the message.
																TRUE = individual_reset *)
    machine_reaction:		machine_reaction_enum;			(* Machine stop type.(emergency, normal,
																on phase, ...) *)
    typology:				message_typology_enum;			(* <a href="#message_typology_enum"><i>typology</i></a> *)	
END_VAR

VAR_IN_OUT
    process:                process;                    	(*$ <a href="#process_object"><i>process</i></a> membership $*)
	CONVERSION_this:		csp_main_motorization_snapshot;			
END_VAR

process_message_init(
	object_name 		:= message_name,
	behaviour 			:= behaviour,
	reset_timeout 		:= reset_timeout,
	disableable 		:= disableable,
	individual_reset 	:= individual_reset,
	machine_reaction 	:= machine_reaction,
	typology			:= typology,
	process 			:= process,
	CONVERSION_this 	:= CONVERSION_this.message);

CONVERSION_this.reason := '';
CONVERSION_this.connection_status := 0;

END_FUNCTION

// ---- Application/CSP/Customer Interface/csp_customerInterfaces.TcPOU
 (*********************************** G.D S.p.A. - Technical Department ***********************************
============= PROGRAM INFO ============
FOLDER:             TBD
MACHINES INVOLVED:  TBD 

============= DESCRIPTION =============
Exit unit device declaration

============= REVISIONS ===============
Date		Version	 	Author      	Description             
----------	-------		------------  	--------------------------------------------
2019/03/27 	0000.00	 	CEC 			Creation of the PRG

**********************************************************************************************************)
(*$R process_ref:= prc; $*)

PROGRAM csp_customerInterfaces

VAR
	prc:								process;
	prc_path:							STRING;
	
	Palletizer:							csp_customerInterfaces_palletizer;
	
END_VAR

VAR PERSISTENT
	CasePacker:							csp_customerInterfaces_casePacker;	
	Order:								csp_customerInterfaces_order;
	Product:							csp_customerInterfaces_product;
	Recipe:								csp_customerInterfaces_recipe;														
	Material:							ARRAY [0..14] OF csp_customerInterfaces_material;
	Mark:								csp_customerInterfaces_mark;
	NextOrder:							csp_customerInterfaces_order;	
	NextProduct:						csp_customerInterfaces_product;	
	NextRecipe:							csp_customerInterfaces_recipe;		
	NextMaterial:						ARRAY [0..14] OF csp_customerInterfaces_material;			
	MES:								csp_customerInterfaces_MES;	
		
END_VAR

_read_var_input();

_objects_manager();

IF NOT objects_running()
THEN
	RETURN;	
END_IF

_read_process_image();

_mode_manager();

CASE process_get_mode(prc) of
	MODE_ABSENT,
	MODE_INACTIVE:
		RETURN;
	MODE_TEST:
		_handle_process_test();
END_CASE

_set_runtime_properties();

(********************************* BODY *********************************)


(* CSP STATUS *)

Dock();
//CasePacker.Status.Online := machine_is_operational(csp.mch); 
//CasePacker.Status.Job := csp_main_brand.p_carton_format;
//CasePacker.Status.NextJob := // need to figure out next job
//CasePacker.Status.Running := machine_is_running(csp.mch);

//**************Variables controlled in csp_main_phaseManager.variables_update******************************

(*CasePacker.Status.Faulted.Main := machine_is_stopped(csp.mch)
									AND csp_main_interface.alarm_id_from_python <> 431 // CYCLE STOP FOR CASE SIDE
									AND csp_main_interface.alarm_id_from_python <> 769; // CYCLE STOP FOR TRANSFER SIDE*)
//CasePacker.Status.Faulted.CaseBlanks := csp_case_feed_magazine.AML_Faulted;

//CasePacker.Status.RunOut := csp_main_motorization.empty_command;
//CasePacker.Status.RunOutComplete := message_is_on(csp_case_virtualMaster.runout_complete);

